(* Schneider Machine Expert - Basic project AWGC_PRODUKSI_TM221CE24R, file version 3.0.0.0 *)
(* ProjectInformations: Name=New project *)

HARDWARE
  Cpu 0: TM221CE24R
  ModuleExtensionObject 0: TM3DI32K
  ModuleExtensionObject 1: TM3AI2H/G
  EthernetConfiguration: NetworkName=M221, IpAllocationMode=FixedAddress, IpAddress=0.0.0.0, SubnetMask=0.0.0.0
  SerialLineConfiguration: Baud=Baud19200, Parity=ParityEven, DataBits=DataBits8, StopBits=StopBits1, PhysicalMedium=PhysicalMediumRs485, TransmissionMode=TransmissionModeModbusRtu, SlaveId=1, Addressing=SlaveAddressing
  MastTask: UsePeriodScanMode=false, PeriodScan=100
  FastTask: Period=255
  CpuBehavior: StartingMode=StartAsPreviousState, AutoSaveRamOnEeprom=true, WatchdogPeriod=250

SYMBOLS  (address, symbol, comment, settings)
  %M0       SYSTEM_ENABLE  "Izin umum gerak"
  %M1       WATER_FAULT  "Fault sinyal level"
  %M2       FAULT_G1  "Fault pintu 1"
  %M3       FAULT_G2  "Fault pintu 2"
  %M4       FAULT_G3  "Fault pintu 3"
  %M5       COMMISSIONING_OK  "Set 1 setelah wiring dan proteksi diuji"
  %M10      REVERSE_G1  "Arah encoder pintu 1 dibalik"
  %M11      REVERSE_G2  "Arah encoder pintu 2 dibalik"
  %M12      REVERSE_G3  "Arah encoder pintu 3 dibalik"
  %M100     G1_BIN_B0  "Binary bit 0 hasil Gray pintu 1"
  %M101     G1_BIN_B1  "Binary bit 1 hasil Gray pintu 1"
  %M102     G1_BIN_B2  "Binary bit 2 hasil Gray pintu 1"
  %M103     G1_BIN_B3  "Binary bit 3 hasil Gray pintu 1"
  %M104     G1_BIN_B4  "Binary bit 4 hasil Gray pintu 1"
  %M105     G1_BIN_B5  "Binary bit 5 hasil Gray pintu 1"
  %M106     G1_BIN_B6  "Binary bit 6 hasil Gray pintu 1"
  %M107     G1_BIN_B7  "Binary bit 7 hasil Gray pintu 1"
  %M110     G2_BIN_B0  "Binary bit 0 hasil Gray pintu 2"
  %M111     G2_BIN_B1  "Binary bit 1 hasil Gray pintu 2"
  %M112     G2_BIN_B2  "Binary bit 2 hasil Gray pintu 2"
  %M113     G2_BIN_B3  "Binary bit 3 hasil Gray pintu 2"
  %M114     G2_BIN_B4  "Binary bit 4 hasil Gray pintu 2"
  %M115     G2_BIN_B5  "Binary bit 5 hasil Gray pintu 2"
  %M116     G2_BIN_B6  "Binary bit 6 hasil Gray pintu 2"
  %M117     G2_BIN_B7  "Binary bit 7 hasil Gray pintu 2"
  %M120     G3_BIN_B0  "Binary bit 0 hasil Gray pintu 3"
  %M121     G3_BIN_B1  "Binary bit 1 hasil Gray pintu 3"
  %M122     G3_BIN_B2  "Binary bit 2 hasil Gray pintu 3"
  %M123     G3_BIN_B3  "Binary bit 3 hasil Gray pintu 3"
  %M124     G3_BIN_B4  "Binary bit 4 hasil Gray pintu 3"
  %M125     G3_BIN_B5  "Binary bit 5 hasil Gray pintu 3"
  %M126     G3_BIN_B6  "Binary bit 6 hasil Gray pintu 3"
  %M127     G3_BIN_B7  "Binary bit 7 hasil Gray pintu 3"
  %M200     AUTO_OPEN_REQ_G1  "Request auto buka G1"
  %M201     AUTO_CLOSE_REQ_G1  "Request auto tutup G1"
  %M202     AUTO_OPEN_REQ_G2  "Request auto buka G2"
  %M203     AUTO_CLOSE_REQ_G2  "Request auto tutup G2"
  %M204     AUTO_OPEN_REQ_G3  "Request auto buka G3"
  %M205     AUTO_CLOSE_REQ_G3  "Request auto tutup G3"
  %M210     MAN_OPEN_REQ_G1  "Request manual buka G1"
  %M211     MAN_CLOSE_REQ_G1  "Request manual tutup G1"
  %M212     MAN_OPEN_REQ_G2  "Request manual buka G2"
  %M213     MAN_CLOSE_REQ_G2  "Request manual tutup G2"
  %M214     MAN_OPEN_REQ_G3  "Request manual buka G3"
  %M215     MAN_CLOSE_REQ_G3  "Request manual tutup G3"
  %M6       SCADA_STOP  "BOOL RW: 1=STOP, 0=release stop; reset to STOP on first RUN"
  %M300     STATUS_I0_0  "Read-only mirror of physical input %I0.0"
  %M301     STATUS_I0_1  "Read-only mirror of physical input %I0.1"
  %M302     STATUS_I0_2  "Read-only mirror of physical input %I0.2"
  %M303     STATUS_I0_3  "Read-only mirror of physical input %I0.3"
  %M304     STATUS_I0_4  "Read-only mirror of physical input %I0.4"
  %M305     STATUS_I0_5  "Read-only mirror of physical input %I0.5"
  %M306     STATUS_I0_6  "Read-only mirror of physical input %I0.6"
  %M307     STATUS_I0_7  "Read-only mirror of physical input %I0.7"
  %M308     STATUS_I0_8  "Read-only mirror of physical input %I0.8"
  %M309     STATUS_I0_9  "Read-only mirror of physical input %I0.9"
  %M310     STATUS_I0_10  "Read-only mirror of physical input %I0.10"
  %M311     STATUS_I0_11  "Read-only mirror of physical input %I0.11"
  %M312     STATUS_I0_12  "Read-only mirror of physical input %I0.12"
  %M313     STATUS_I0_13  "Read-only mirror of physical input %I0.13"
  %M344     STATUS_I1_24  "Read-only mirror of physical input %I1.24"
  %M345     STATUS_I1_25  "Read-only mirror of physical input %I1.25"
  %M346     STATUS_I1_26  "Read-only mirror of physical input %I1.26"
  %M347     STATUS_I1_27  "Read-only mirror of physical input %I1.27"
  %M348     STATUS_I1_28  "Read-only mirror of physical input %I1.28"
  %M349     STATUS_I1_29  "Read-only mirror of physical input %I1.29"
  %M350     STATUS_I1_30  "Read-only mirror of physical input %I1.30"
  %M351     STATUS_I1_31  "Read-only mirror of physical input %I1.31"
  %M360     STATUS_Q0_0  "Read-only mirror of actual output %Q0.0"
  %M361     STATUS_Q0_1  "Read-only mirror of actual output %Q0.1"
  %M362     STATUS_Q0_2  "Read-only mirror of actual output %Q0.2"
  %M363     STATUS_Q0_3  "Read-only mirror of actual output %Q0.3"
  %M364     STATUS_Q0_4  "Read-only mirror of actual output %Q0.4"
  %M365     STATUS_Q0_5  "Read-only mirror of actual output %Q0.5"
  %S13      SB_FIRSTRUN  "Indicates the first controller cycle in RUN mode"
  %MW1      WATER_RANGE_MM  "Range sensor level mm"
  %MW2      LEVEL_RAW_COPY  "Salinan raw input level"
  %MW10     MAX_HEIGHT_G1_MM  "Tinggi maksimum pintu 1 mm"
  %MW11     MAX_HEIGHT_G2_MM  "Tinggi maksimum pintu 2 mm"
  %MW12     MAX_HEIGHT_G3_MM  "Tinggi maksimum pintu 3 mm"
  %MW13     DEADBAND_PCT  "Deadband posisi persen"
  %MW20     ENC_ZERO_G1  "Nilai encoder pintu 1 saat tertutup"
  %MW21     ENC_ZERO_G2  "Nilai encoder pintu 2 saat tertutup"
  %MW22     ENC_ZERO_G3  "Nilai encoder pintu 3 saat tertutup"
  %MW23     ENC_SPAN_G1  "Span count tertutup-terbuka G1"
  %MW24     ENC_SPAN_G2  "Span count tertutup-terbuka G2"
  %MW25     ENC_SPAN_G3  "Span count tertutup-terbuka G3"
  %MW30     ENC_BINARY_G1  "Nilai biner encoder G1"
  %MW31     ENC_BINARY_G2  "Nilai biner encoder G2"
  %MW32     ENC_BINARY_G3  "Nilai biner encoder G3"
  %MW33     POS_COUNT_G1  "Count posisi terkoreksi G1"
  %MW34     POS_COUNT_G2  "Count posisi terkoreksi G2"
  %MW35     POS_COUNT_G3  "Count posisi terkoreksi G3"
  %MW50     TARGET_PCT_G1  "Target bukaan G1 0-100 persen"
  %MW51     TARGET_PCT_G2  "Target bukaan G2 0-100 persen"
  %MW52     TARGET_PCT_G3  "Target bukaan G3 0-100 persen"
  %MW110    SCADA_PROFILE_ID  "221 identifies AWGC SCADA map"
  %MW111    SCADA_PROFILE_VERSION  "3001 production profile: physical inputs and relay outputs"
  %MF60     POSITION_G1_PCT  "Posisi G1 persen"
  %MF62     POSITION_G2_PCT  "Posisi G2 persen"
  %MF64     POSITION_G3_PCT  "Posisi G3 persen"
  %MF66     POSITION_G1_MM  "Posisi G1 mm"
  %MF68     POSITION_G2_MM  "Posisi G2 mm"
  %MF70     POSITION_G3_MM  "Posisi G3 mm"
  %MF72     WATER_LEVEL_MM  "Level air mm"
  %MF74     WATER_LEVEL_PCT  "Level air persen"
  %MF76     WATER_RANGE_REAL  "Range level dalam REAL"
  %MF80     TARGET_G1_REAL  "Target G1 dalam REAL"
  %MF82     TARGET_G2_REAL  "Target G2 dalam REAL"
  %MF84     TARGET_G3_REAL  "Target G3 dalam REAL"
  %MF86     DEADBAND_REAL  "Deadband dalam REAL"
  %MF88     OPEN_THRESHOLD_G1  "Ambang buka G1"
  %MF90     CLOSE_THRESHOLD_G1  "Ambang tutup G1"
  %MF92     OPEN_THRESHOLD_G2  "Ambang buka G2"
  %MF94     CLOSE_THRESHOLD_G2  "Ambang tutup G2"
  %MF96     OPEN_THRESHOLD_G3  "Ambang buka G3"
  %MF98     CLOSE_THRESHOLD_G3  "Ambang tutup G3"
  %I0.0     SAFETY_OK_IN  "Feedback rangkaian safety hardwired sehat"
  %I0.1     LS_CLOSE_G1  "Limit tertutup pintu 1"
  %I0.2     LS_OPEN_G1  "Limit terbuka pintu 1"
  %I0.3     LS_CLOSE_G2  "Limit tertutup pintu 2"
  %I0.4     LS_OPEN_G2  "Limit terbuka pintu 2"
  %I0.5     LS_CLOSE_G3  "Limit tertutup pintu 3"
  %I0.6     LS_OPEN_G3  "Limit terbuka pintu 3"
  %I0.7     OL_OK_G1  "Overload motor pintu 1 sehat"
  %I0.8     OL_OK_G2  "Overload motor pintu 2 sehat"
  %I0.9     OL_OK_G3  "Overload motor pintu 3 sehat"
  %I0.10    SPARE_I010  "Cadangan input"
  %I0.11    SPARE_I011  "Cadangan input"
  %I0.12    SPARE_I012  "Cadangan input"
  %I0.13    SPARE_I013  "Cadangan input"
  %Q0.0     OPEN_G1  "Relay kontaktor OPEN pintu 1"
  %Q0.1     CLOSE_G1  "Relay kontaktor CLOSE pintu 1"
  %Q0.2     OPEN_G2  "Relay kontaktor OPEN pintu 2"
  %Q0.3     CLOSE_G2  "Relay kontaktor CLOSE pintu 2"
  %Q0.4     OPEN_G3  "Relay kontaktor OPEN pintu 3"
  %Q0.5     CLOSE_G3  "Relay kontaktor CLOSE pintu 3"
  %I1.0     ENC_G1_GRAY_B0  "E6CP pintu 1 Gray bit 0"
  %I1.1     ENC_G1_GRAY_B1  "E6CP pintu 1 Gray bit 1"
  %I1.2     ENC_G1_GRAY_B2  "E6CP pintu 1 Gray bit 2"
  %I1.3     ENC_G1_GRAY_B3  "E6CP pintu 1 Gray bit 3"
  %I1.4     ENC_G1_GRAY_B4  "E6CP pintu 1 Gray bit 4"
  %I1.5     ENC_G1_GRAY_B5  "E6CP pintu 1 Gray bit 5"
  %I1.6     ENC_G1_GRAY_B6  "E6CP pintu 1 Gray bit 6"
  %I1.7     ENC_G1_GRAY_B7  "E6CP pintu 1 Gray bit 7"
  %I1.8     ENC_G2_GRAY_B0  "E6CP pintu 2 Gray bit 0"
  %I1.9     ENC_G2_GRAY_B1  "E6CP pintu 2 Gray bit 1"
  %I1.10    ENC_G2_GRAY_B2  "E6CP pintu 2 Gray bit 2"
  %I1.11    ENC_G2_GRAY_B3  "E6CP pintu 2 Gray bit 3"
  %I1.12    ENC_G2_GRAY_B4  "E6CP pintu 2 Gray bit 4"
  %I1.13    ENC_G2_GRAY_B5  "E6CP pintu 2 Gray bit 5"
  %I1.14    ENC_G2_GRAY_B6  "E6CP pintu 2 Gray bit 6"
  %I1.15    ENC_G2_GRAY_B7  "E6CP pintu 2 Gray bit 7"
  %I1.16    ENC_G3_GRAY_B0  "E6CP pintu 3 Gray bit 0"
  %I1.17    ENC_G3_GRAY_B1  "E6CP pintu 3 Gray bit 1"
  %I1.18    ENC_G3_GRAY_B2  "E6CP pintu 3 Gray bit 2"
  %I1.19    ENC_G3_GRAY_B3  "E6CP pintu 3 Gray bit 3"
  %I1.20    ENC_G3_GRAY_B4  "E6CP pintu 3 Gray bit 4"
  %I1.21    ENC_G3_GRAY_B5  "E6CP pintu 3 Gray bit 5"
  %I1.22    ENC_G3_GRAY_B6  "E6CP pintu 3 Gray bit 6"
  %I1.23    ENC_G3_GRAY_B7  "E6CP pintu 3 Gray bit 7"
  %I1.24    MODE_AUTO  "Selector 1=AUTO 0=MANUAL"
  %I1.25    MAN_OPEN_G1  "PB manual buka pintu 1"
  %I1.26    MAN_CLOSE_G1  "PB manual tutup pintu 1"
  %I1.27    MAN_OPEN_G2  "PB manual buka pintu 2"
  %I1.28    MAN_CLOSE_G2  "PB manual tutup pintu 2"
  %I1.29    MAN_OPEN_G3  "PB manual buka pintu 3"
  %I1.30    MAN_CLOSE_G3  "PB manual tutup pintu 3"
  %I1.31    RESET_FAULT  "PB reset fault"
  %IW2.0    LEVEL_RAW  "Sensor level 4-20 mA raw 4000-20000"  [Type=Type_4_20mA, Scope=Scope_Customized, Minimum=4000, Maximum=20000]

POU AWGC_3_PINTU_IL
  (* SectionNumber=1 *)

// Rung 0: REV3_SCADA_VERSION
// SCADA compatibility marker for production profile.
  LD 1
  [ %MW111 := 3001 ]      (* SCADA_PROFILE_VERSION *)
  // as ST:
  //   SCADA_PROFILE_VERSION := 3001;

// Rung 1: REV3_SCADA_ID
// SCADA compatibility marker for production profile.
  LD 1
  [ %MW110 := 221 ]       (* SCADA_PROFILE_ID *)
  // as ST:
  //   SCADA_PROFILE_ID := 221;

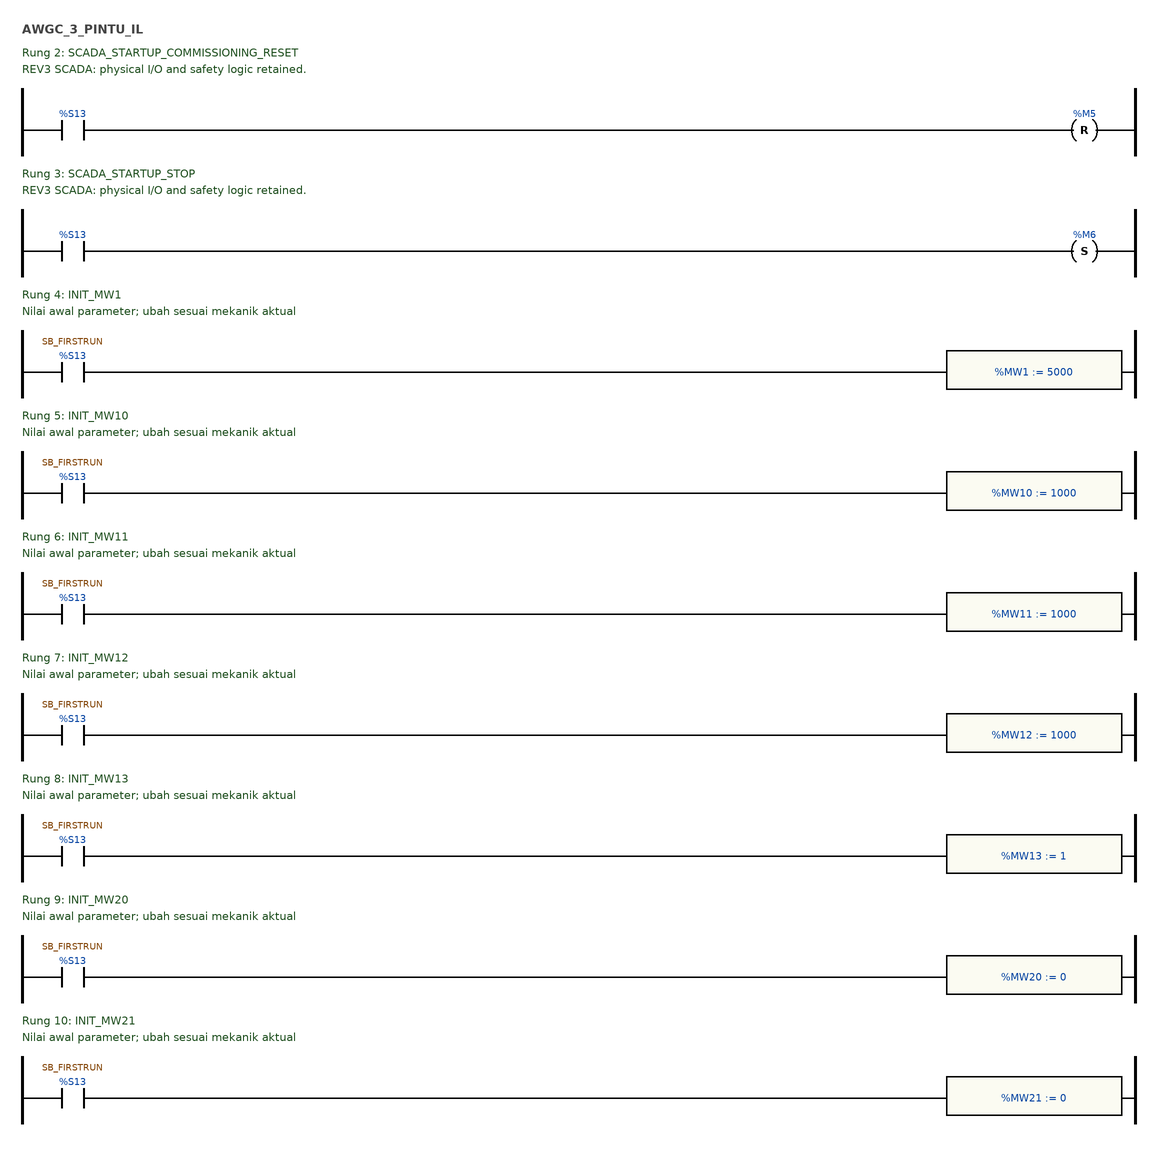

// Rung 2: SCADA_STARTUP_COMMISSIONING_RESET
// REV3 SCADA: physical I/O and safety logic retained.
  LD %S13                 (* SB_FIRSTRUN *)
  R %M5                   (* COMMISSIONING_OK *)
  // as ST:
  //   IF SB_FIRSTRUN THEN COMMISSIONING_OK := FALSE; END_IF;

// Rung 3: SCADA_STARTUP_STOP
// REV3 SCADA: physical I/O and safety logic retained.
  LD %S13                 (* SB_FIRSTRUN *)
  S %M6                   (* SCADA_STOP *)
  // as ST:
  //   IF SB_FIRSTRUN THEN SCADA_STOP := TRUE; END_IF;

// Rung 4: INIT_MW1
// Nilai awal parameter; ubah sesuai mekanik aktual
  LD %S13                 (* SB_FIRSTRUN *)
  [ %MW1 := 5000 ]        (* WATER_RANGE_MM *)
  // as ST:
  //   IF SB_FIRSTRUN THEN WATER_RANGE_MM := 5000; END_IF;

// Rung 5: INIT_MW10
// Nilai awal parameter; ubah sesuai mekanik aktual
  LD %S13                 (* SB_FIRSTRUN *)
  [ %MW10 := 1000 ]       (* MAX_HEIGHT_G1_MM *)
  // as ST:
  //   IF SB_FIRSTRUN THEN MAX_HEIGHT_G1_MM := 1000; END_IF;

// Rung 6: INIT_MW11
// Nilai awal parameter; ubah sesuai mekanik aktual
  LD %S13                 (* SB_FIRSTRUN *)
  [ %MW11 := 1000 ]       (* MAX_HEIGHT_G2_MM *)
  // as ST:
  //   IF SB_FIRSTRUN THEN MAX_HEIGHT_G2_MM := 1000; END_IF;

// Rung 7: INIT_MW12
// Nilai awal parameter; ubah sesuai mekanik aktual
  LD %S13                 (* SB_FIRSTRUN *)
  [ %MW12 := 1000 ]       (* MAX_HEIGHT_G3_MM *)
  // as ST:
  //   IF SB_FIRSTRUN THEN MAX_HEIGHT_G3_MM := 1000; END_IF;

// Rung 8: INIT_MW13
// Nilai awal parameter; ubah sesuai mekanik aktual
  LD %S13                 (* SB_FIRSTRUN *)
  [ %MW13 := 1 ]          (* DEADBAND_PCT *)
  // as ST:
  //   IF SB_FIRSTRUN THEN DEADBAND_PCT := 1; END_IF;

// Rung 9: INIT_MW20
// Nilai awal parameter; ubah sesuai mekanik aktual
  LD %S13                 (* SB_FIRSTRUN *)
  [ %MW20 := 0 ]          (* ENC_ZERO_G1 *)
  // as ST:
  //   IF SB_FIRSTRUN THEN ENC_ZERO_G1 := 0; END_IF;

// Rung 10: INIT_MW21
// Nilai awal parameter; ubah sesuai mekanik aktual
  LD %S13                 (* SB_FIRSTRUN *)
  [ %MW21 := 0 ]          (* ENC_ZERO_G2 *)
  // as ST:
  //   IF SB_FIRSTRUN THEN ENC_ZERO_G2 := 0; END_IF;

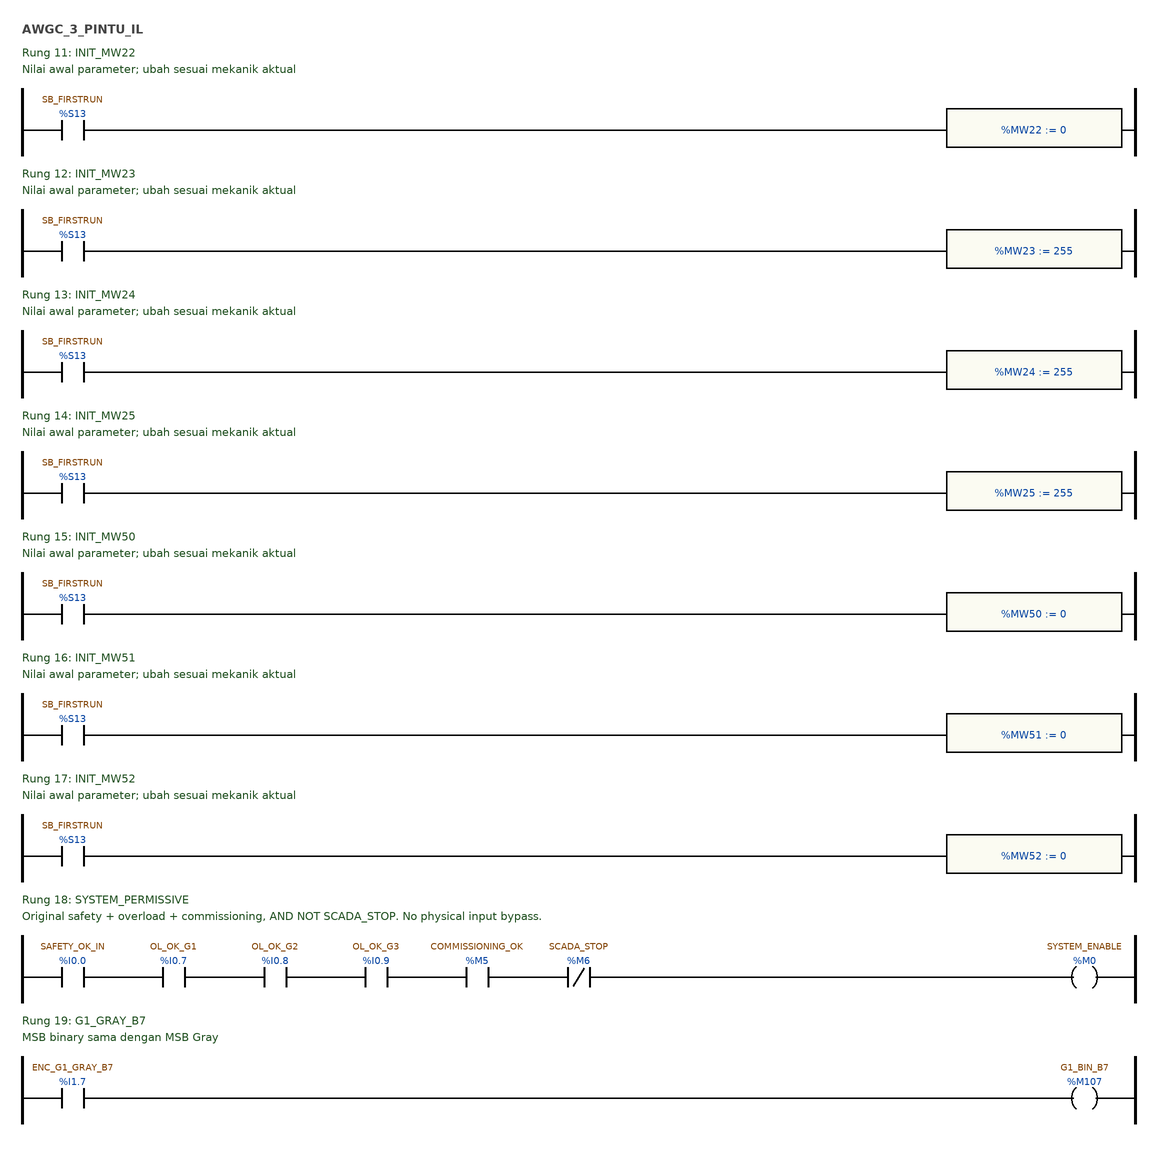

// Rung 11: INIT_MW22
// Nilai awal parameter; ubah sesuai mekanik aktual
  LD %S13                 (* SB_FIRSTRUN *)
  [ %MW22 := 0 ]          (* ENC_ZERO_G3 *)
  // as ST:
  //   IF SB_FIRSTRUN THEN ENC_ZERO_G3 := 0; END_IF;

// Rung 12: INIT_MW23
// Nilai awal parameter; ubah sesuai mekanik aktual
  LD %S13                 (* SB_FIRSTRUN *)
  [ %MW23 := 255 ]        (* ENC_SPAN_G1 *)
  // as ST:
  //   IF SB_FIRSTRUN THEN ENC_SPAN_G1 := 255; END_IF;

// Rung 13: INIT_MW24
// Nilai awal parameter; ubah sesuai mekanik aktual
  LD %S13                 (* SB_FIRSTRUN *)
  [ %MW24 := 255 ]        (* ENC_SPAN_G2 *)
  // as ST:
  //   IF SB_FIRSTRUN THEN ENC_SPAN_G2 := 255; END_IF;

// Rung 14: INIT_MW25
// Nilai awal parameter; ubah sesuai mekanik aktual
  LD %S13                 (* SB_FIRSTRUN *)
  [ %MW25 := 255 ]        (* ENC_SPAN_G3 *)
  // as ST:
  //   IF SB_FIRSTRUN THEN ENC_SPAN_G3 := 255; END_IF;

// Rung 15: INIT_MW50
// Nilai awal parameter; ubah sesuai mekanik aktual
  LD %S13                 (* SB_FIRSTRUN *)
  [ %MW50 := 0 ]          (* TARGET_PCT_G1 *)
  // as ST:
  //   IF SB_FIRSTRUN THEN TARGET_PCT_G1 := 0; END_IF;

// Rung 16: INIT_MW51
// Nilai awal parameter; ubah sesuai mekanik aktual
  LD %S13                 (* SB_FIRSTRUN *)
  [ %MW51 := 0 ]          (* TARGET_PCT_G2 *)
  // as ST:
  //   IF SB_FIRSTRUN THEN TARGET_PCT_G2 := 0; END_IF;

// Rung 17: INIT_MW52
// Nilai awal parameter; ubah sesuai mekanik aktual
  LD %S13                 (* SB_FIRSTRUN *)
  [ %MW52 := 0 ]          (* TARGET_PCT_G3 *)
  // as ST:
  //   IF SB_FIRSTRUN THEN TARGET_PCT_G3 := 0; END_IF;

// Rung 18: SYSTEM_PERMISSIVE
// Original safety + overload + commissioning, AND NOT SCADA_STOP. No physical input bypass.
  LD %I0.0                (* SAFETY_OK_IN *)
  AND %I0.7               (* OL_OK_G1 *)
  AND %I0.8               (* OL_OK_G2 *)
  AND %I0.9               (* OL_OK_G3 *)
  AND %M5                 (* COMMISSIONING_OK *)
  ANDN %M6                (* SCADA_STOP *)
  ST %M0                  (* SYSTEM_ENABLE *)
  // %M6: 1=STOP; startup STOP. This is not an emergency stop.
  // as ST:
  //   SYSTEM_ENABLE := SAFETY_OK_IN AND OL_OK_G1 AND OL_OK_G2 AND OL_OK_G3 AND COMMISSIONING_OK AND NOT SCADA_STOP;

// Rung 19: G1_GRAY_B7
// MSB binary sama dengan MSB Gray
  LD %I1.7                (* ENC_G1_GRAY_B7 *)
  ST %M107                (* G1_BIN_B7 *)
  // as ST:
  //   G1_BIN_B7 := ENC_G1_GRAY_B7;

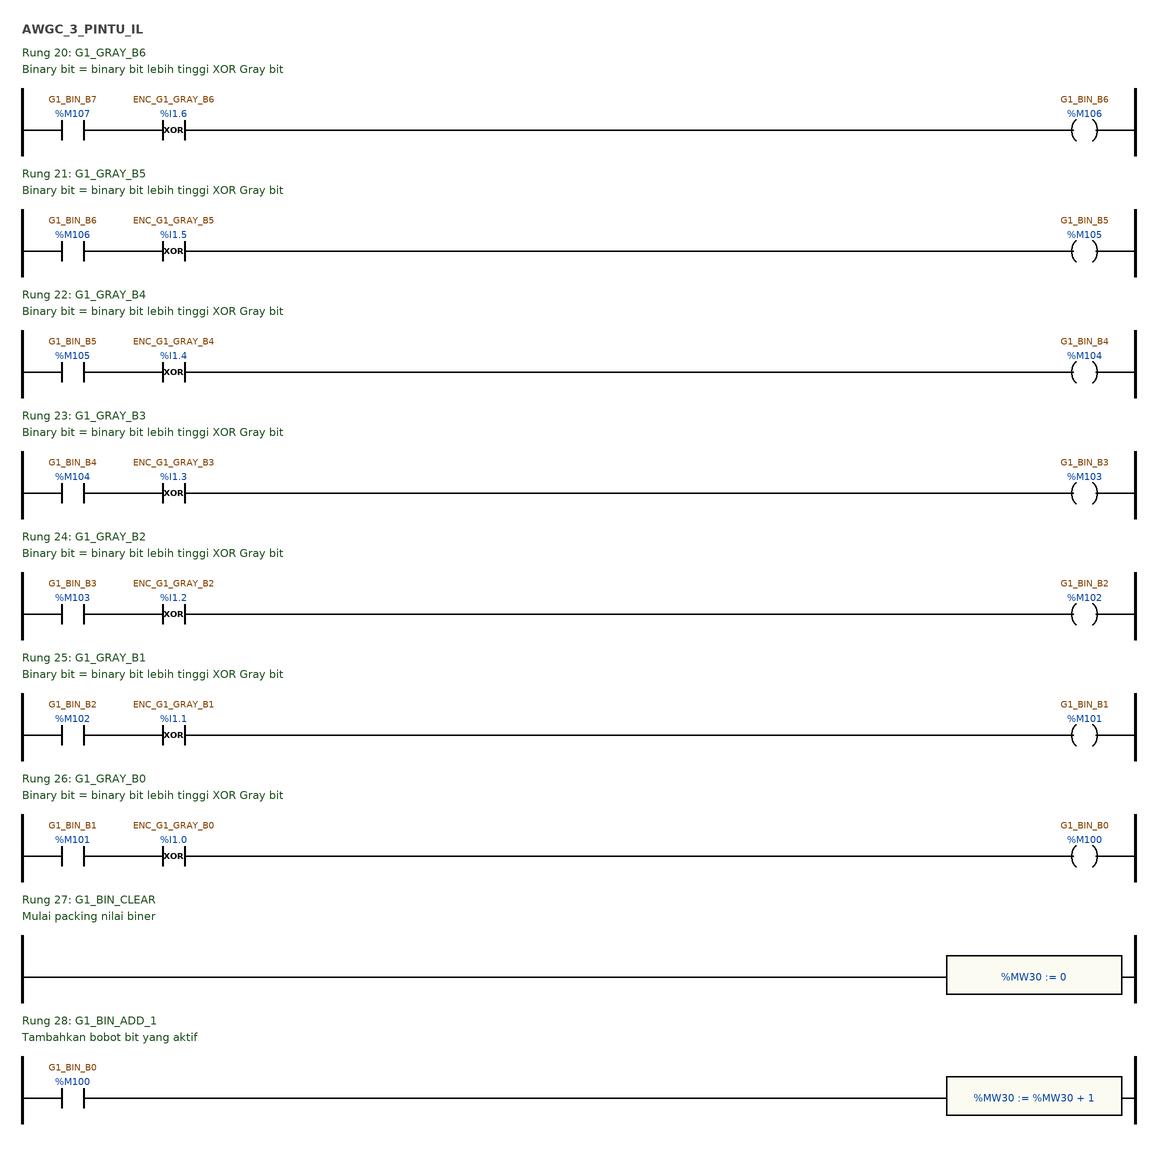

// Rung 20: G1_GRAY_B6
// Binary bit = binary bit lebih tinggi XOR Gray bit
  LD %M107                (* G1_BIN_B7 *)
  XOR %I1.6               (* ENC_G1_GRAY_B6 *)
  ST %M106                (* G1_BIN_B6 *)
  // as ST:
  //   G1_BIN_B6 := G1_BIN_B7 XOR ENC_G1_GRAY_B6;

// Rung 21: G1_GRAY_B5
// Binary bit = binary bit lebih tinggi XOR Gray bit
  LD %M106                (* G1_BIN_B6 *)
  XOR %I1.5               (* ENC_G1_GRAY_B5 *)
  ST %M105                (* G1_BIN_B5 *)
  // as ST:
  //   G1_BIN_B5 := G1_BIN_B6 XOR ENC_G1_GRAY_B5;

// Rung 22: G1_GRAY_B4
// Binary bit = binary bit lebih tinggi XOR Gray bit
  LD %M105                (* G1_BIN_B5 *)
  XOR %I1.4               (* ENC_G1_GRAY_B4 *)
  ST %M104                (* G1_BIN_B4 *)
  // as ST:
  //   G1_BIN_B4 := G1_BIN_B5 XOR ENC_G1_GRAY_B4;

// Rung 23: G1_GRAY_B3
// Binary bit = binary bit lebih tinggi XOR Gray bit
  LD %M104                (* G1_BIN_B4 *)
  XOR %I1.3               (* ENC_G1_GRAY_B3 *)
  ST %M103                (* G1_BIN_B3 *)
  // as ST:
  //   G1_BIN_B3 := G1_BIN_B4 XOR ENC_G1_GRAY_B3;

// Rung 24: G1_GRAY_B2
// Binary bit = binary bit lebih tinggi XOR Gray bit
  LD %M103                (* G1_BIN_B3 *)
  XOR %I1.2               (* ENC_G1_GRAY_B2 *)
  ST %M102                (* G1_BIN_B2 *)
  // as ST:
  //   G1_BIN_B2 := G1_BIN_B3 XOR ENC_G1_GRAY_B2;

// Rung 25: G1_GRAY_B1
// Binary bit = binary bit lebih tinggi XOR Gray bit
  LD %M102                (* G1_BIN_B2 *)
  XOR %I1.1               (* ENC_G1_GRAY_B1 *)
  ST %M101                (* G1_BIN_B1 *)
  // as ST:
  //   G1_BIN_B1 := G1_BIN_B2 XOR ENC_G1_GRAY_B1;

// Rung 26: G1_GRAY_B0
// Binary bit = binary bit lebih tinggi XOR Gray bit
  LD %M101                (* G1_BIN_B1 *)
  XOR %I1.0               (* ENC_G1_GRAY_B0 *)
  ST %M100                (* G1_BIN_B0 *)
  // as ST:
  //   G1_BIN_B0 := G1_BIN_B1 XOR ENC_G1_GRAY_B0;

// Rung 27: G1_BIN_CLEAR
// Mulai packing nilai biner
  LD 1
  [ %MW30 := 0 ]          (* ENC_BINARY_G1 *)
  // as ST:
  //   ENC_BINARY_G1 := 0;

// Rung 28: G1_BIN_ADD_1
// Tambahkan bobot bit yang aktif
  LD %M100                (* G1_BIN_B0 *)
  [ %MW30 := %MW30 + 1 ]  (* ENC_BINARY_G1, ENC_BINARY_G1 *)
  // as ST:
  //   IF G1_BIN_B0 THEN ENC_BINARY_G1 := ENC_BINARY_G1 + 1; END_IF;

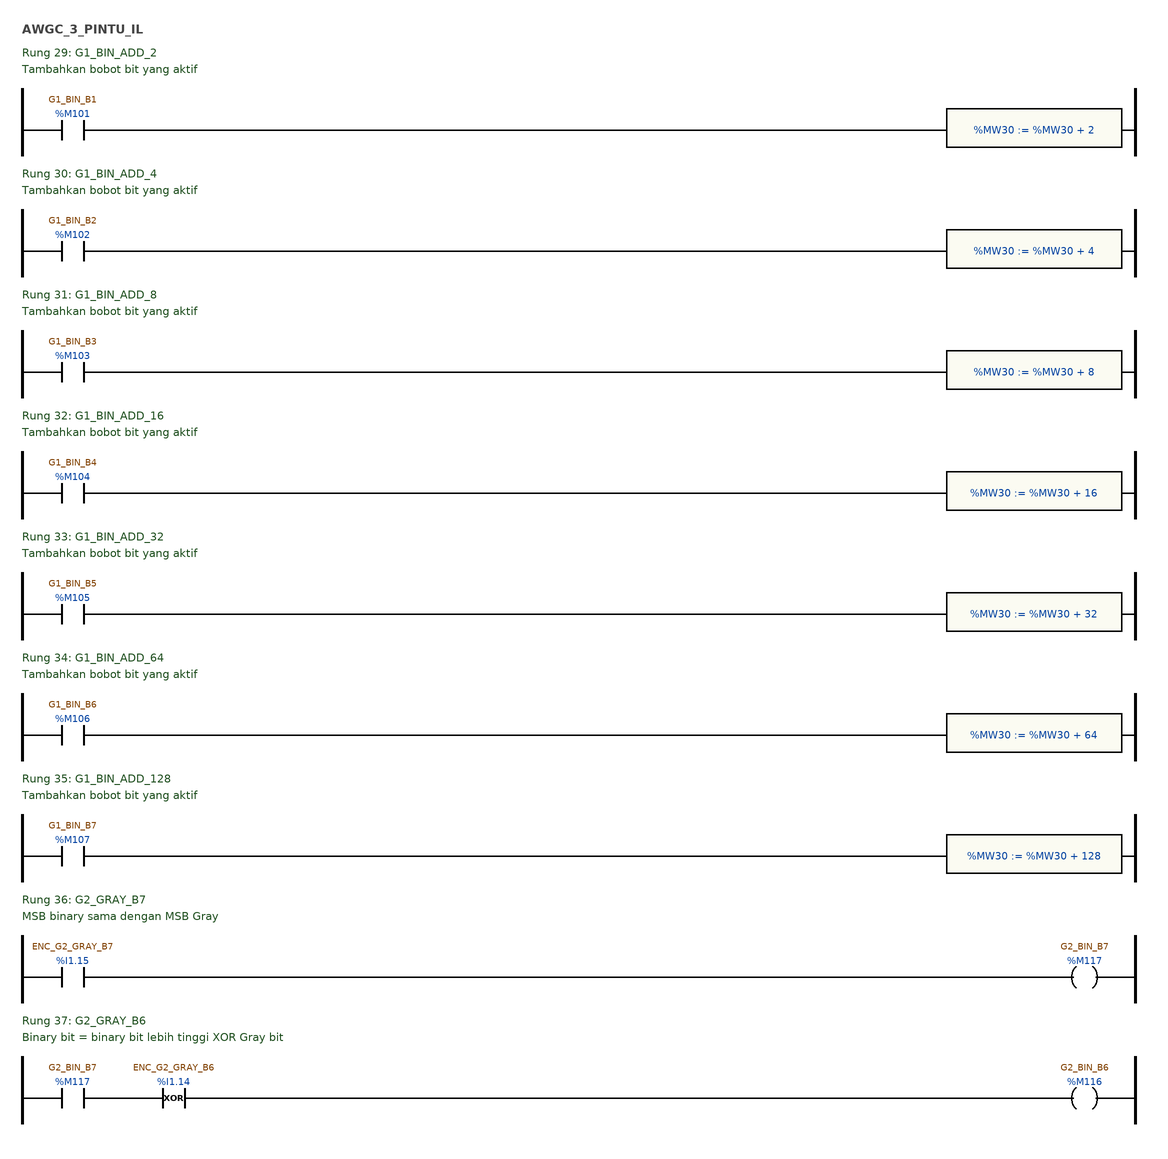

// Rung 29: G1_BIN_ADD_2
// Tambahkan bobot bit yang aktif
  LD %M101                (* G1_BIN_B1 *)
  [ %MW30 := %MW30 + 2 ]  (* ENC_BINARY_G1, ENC_BINARY_G1 *)
  // as ST:
  //   IF G1_BIN_B1 THEN ENC_BINARY_G1 := ENC_BINARY_G1 + 2; END_IF;

// Rung 30: G1_BIN_ADD_4
// Tambahkan bobot bit yang aktif
  LD %M102                (* G1_BIN_B2 *)
  [ %MW30 := %MW30 + 4 ]  (* ENC_BINARY_G1, ENC_BINARY_G1 *)
  // as ST:
  //   IF G1_BIN_B2 THEN ENC_BINARY_G1 := ENC_BINARY_G1 + 4; END_IF;

// Rung 31: G1_BIN_ADD_8
// Tambahkan bobot bit yang aktif
  LD %M103                (* G1_BIN_B3 *)
  [ %MW30 := %MW30 + 8 ]  (* ENC_BINARY_G1, ENC_BINARY_G1 *)
  // as ST:
  //   IF G1_BIN_B3 THEN ENC_BINARY_G1 := ENC_BINARY_G1 + 8; END_IF;

// Rung 32: G1_BIN_ADD_16
// Tambahkan bobot bit yang aktif
  LD %M104                (* G1_BIN_B4 *)
  [ %MW30 := %MW30 + 16 ] (* ENC_BINARY_G1, ENC_BINARY_G1 *)
  // as ST:
  //   IF G1_BIN_B4 THEN ENC_BINARY_G1 := ENC_BINARY_G1 + 16; END_IF;

// Rung 33: G1_BIN_ADD_32
// Tambahkan bobot bit yang aktif
  LD %M105                (* G1_BIN_B5 *)
  [ %MW30 := %MW30 + 32 ] (* ENC_BINARY_G1, ENC_BINARY_G1 *)
  // as ST:
  //   IF G1_BIN_B5 THEN ENC_BINARY_G1 := ENC_BINARY_G1 + 32; END_IF;

// Rung 34: G1_BIN_ADD_64
// Tambahkan bobot bit yang aktif
  LD %M106                (* G1_BIN_B6 *)
  [ %MW30 := %MW30 + 64 ] (* ENC_BINARY_G1, ENC_BINARY_G1 *)
  // as ST:
  //   IF G1_BIN_B6 THEN ENC_BINARY_G1 := ENC_BINARY_G1 + 64; END_IF;

// Rung 35: G1_BIN_ADD_128
// Tambahkan bobot bit yang aktif
  LD %M107                (* G1_BIN_B7 *)
  [ %MW30 := %MW30 + 128 ](* ENC_BINARY_G1, ENC_BINARY_G1 *)
  // as ST:
  //   IF G1_BIN_B7 THEN ENC_BINARY_G1 := ENC_BINARY_G1 + 128; END_IF;

// Rung 36: G2_GRAY_B7
// MSB binary sama dengan MSB Gray
  LD %I1.15               (* ENC_G2_GRAY_B7 *)
  ST %M117                (* G2_BIN_B7 *)
  // as ST:
  //   G2_BIN_B7 := ENC_G2_GRAY_B7;

// Rung 37: G2_GRAY_B6
// Binary bit = binary bit lebih tinggi XOR Gray bit
  LD %M117                (* G2_BIN_B7 *)
  XOR %I1.14              (* ENC_G2_GRAY_B6 *)
  ST %M116                (* G2_BIN_B6 *)
  // as ST:
  //   G2_BIN_B6 := G2_BIN_B7 XOR ENC_G2_GRAY_B6;

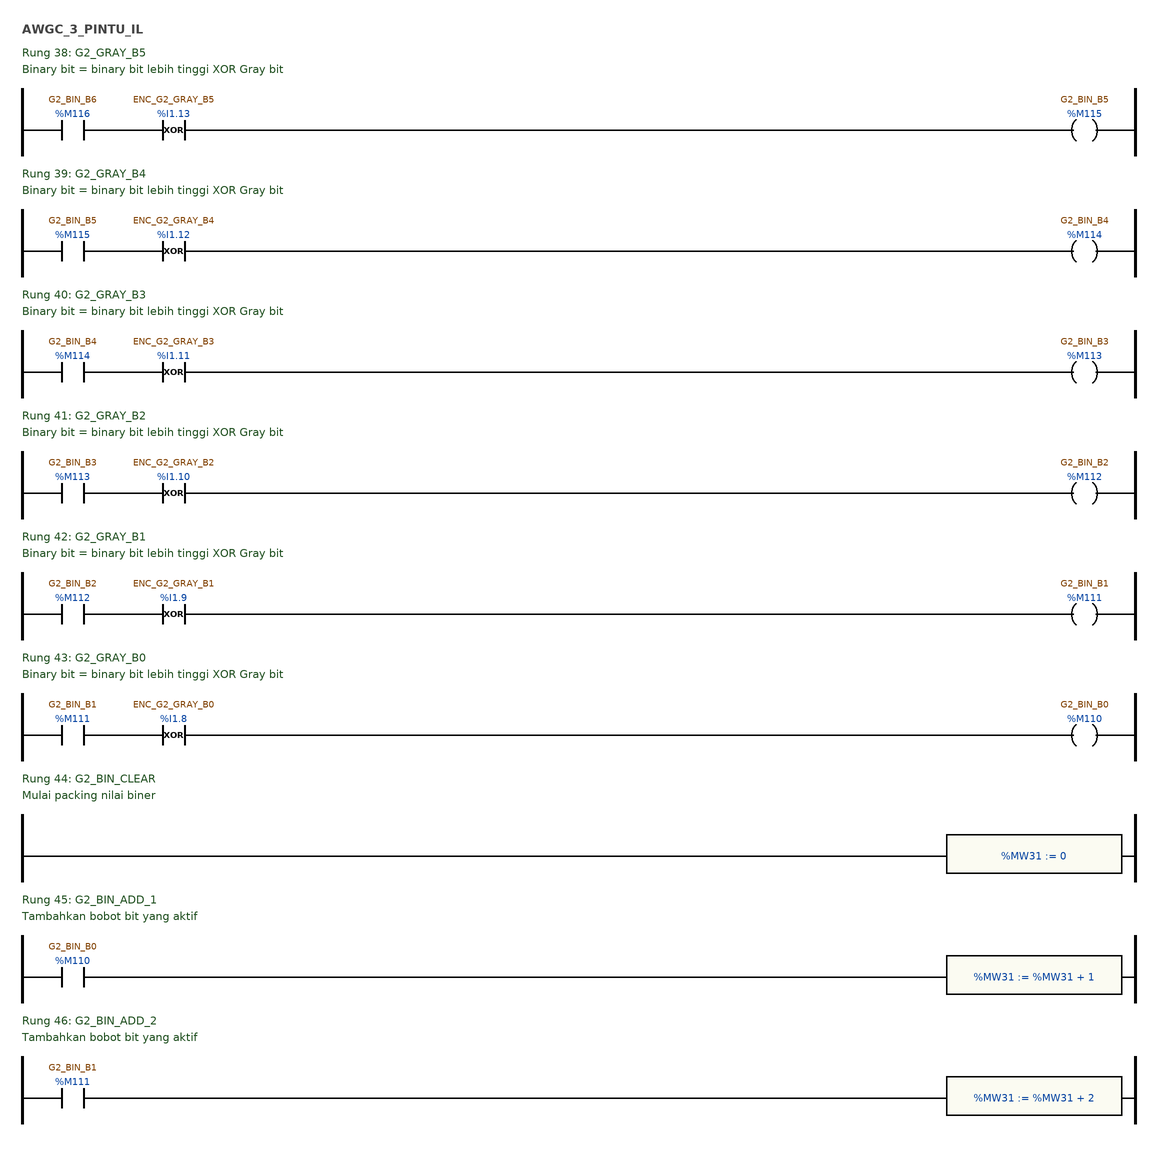

// Rung 38: G2_GRAY_B5
// Binary bit = binary bit lebih tinggi XOR Gray bit
  LD %M116                (* G2_BIN_B6 *)
  XOR %I1.13              (* ENC_G2_GRAY_B5 *)
  ST %M115                (* G2_BIN_B5 *)
  // as ST:
  //   G2_BIN_B5 := G2_BIN_B6 XOR ENC_G2_GRAY_B5;

// Rung 39: G2_GRAY_B4
// Binary bit = binary bit lebih tinggi XOR Gray bit
  LD %M115                (* G2_BIN_B5 *)
  XOR %I1.12              (* ENC_G2_GRAY_B4 *)
  ST %M114                (* G2_BIN_B4 *)
  // as ST:
  //   G2_BIN_B4 := G2_BIN_B5 XOR ENC_G2_GRAY_B4;

// Rung 40: G2_GRAY_B3
// Binary bit = binary bit lebih tinggi XOR Gray bit
  LD %M114                (* G2_BIN_B4 *)
  XOR %I1.11              (* ENC_G2_GRAY_B3 *)
  ST %M113                (* G2_BIN_B3 *)
  // as ST:
  //   G2_BIN_B3 := G2_BIN_B4 XOR ENC_G2_GRAY_B3;

// Rung 41: G2_GRAY_B2
// Binary bit = binary bit lebih tinggi XOR Gray bit
  LD %M113                (* G2_BIN_B3 *)
  XOR %I1.10              (* ENC_G2_GRAY_B2 *)
  ST %M112                (* G2_BIN_B2 *)
  // as ST:
  //   G2_BIN_B2 := G2_BIN_B3 XOR ENC_G2_GRAY_B2;

// Rung 42: G2_GRAY_B1
// Binary bit = binary bit lebih tinggi XOR Gray bit
  LD %M112                (* G2_BIN_B2 *)
  XOR %I1.9               (* ENC_G2_GRAY_B1 *)
  ST %M111                (* G2_BIN_B1 *)
  // as ST:
  //   G2_BIN_B1 := G2_BIN_B2 XOR ENC_G2_GRAY_B1;

// Rung 43: G2_GRAY_B0
// Binary bit = binary bit lebih tinggi XOR Gray bit
  LD %M111                (* G2_BIN_B1 *)
  XOR %I1.8               (* ENC_G2_GRAY_B0 *)
  ST %M110                (* G2_BIN_B0 *)
  // as ST:
  //   G2_BIN_B0 := G2_BIN_B1 XOR ENC_G2_GRAY_B0;

// Rung 44: G2_BIN_CLEAR
// Mulai packing nilai biner
  LD 1
  [ %MW31 := 0 ]          (* ENC_BINARY_G2 *)
  // as ST:
  //   ENC_BINARY_G2 := 0;

// Rung 45: G2_BIN_ADD_1
// Tambahkan bobot bit yang aktif
  LD %M110                (* G2_BIN_B0 *)
  [ %MW31 := %MW31 + 1 ]  (* ENC_BINARY_G2, ENC_BINARY_G2 *)
  // as ST:
  //   IF G2_BIN_B0 THEN ENC_BINARY_G2 := ENC_BINARY_G2 + 1; END_IF;

// Rung 46: G2_BIN_ADD_2
// Tambahkan bobot bit yang aktif
  LD %M111                (* G2_BIN_B1 *)
  [ %MW31 := %MW31 + 2 ]  (* ENC_BINARY_G2, ENC_BINARY_G2 *)
  // as ST:
  //   IF G2_BIN_B1 THEN ENC_BINARY_G2 := ENC_BINARY_G2 + 2; END_IF;

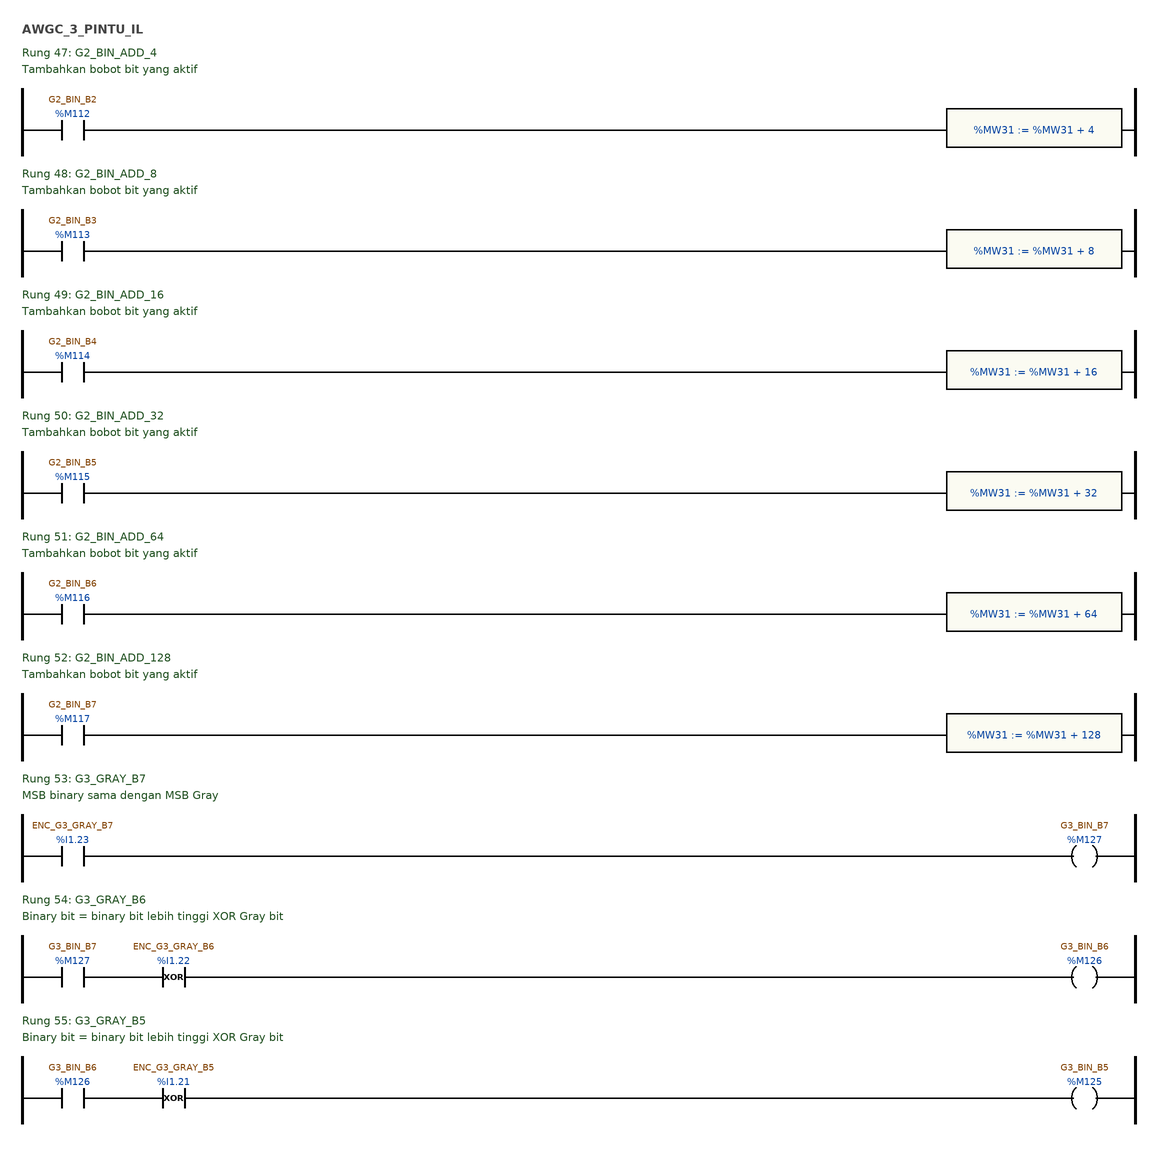

// Rung 47: G2_BIN_ADD_4
// Tambahkan bobot bit yang aktif
  LD %M112                (* G2_BIN_B2 *)
  [ %MW31 := %MW31 + 4 ]  (* ENC_BINARY_G2, ENC_BINARY_G2 *)
  // as ST:
  //   IF G2_BIN_B2 THEN ENC_BINARY_G2 := ENC_BINARY_G2 + 4; END_IF;

// Rung 48: G2_BIN_ADD_8
// Tambahkan bobot bit yang aktif
  LD %M113                (* G2_BIN_B3 *)
  [ %MW31 := %MW31 + 8 ]  (* ENC_BINARY_G2, ENC_BINARY_G2 *)
  // as ST:
  //   IF G2_BIN_B3 THEN ENC_BINARY_G2 := ENC_BINARY_G2 + 8; END_IF;

// Rung 49: G2_BIN_ADD_16
// Tambahkan bobot bit yang aktif
  LD %M114                (* G2_BIN_B4 *)
  [ %MW31 := %MW31 + 16 ] (* ENC_BINARY_G2, ENC_BINARY_G2 *)
  // as ST:
  //   IF G2_BIN_B4 THEN ENC_BINARY_G2 := ENC_BINARY_G2 + 16; END_IF;

// Rung 50: G2_BIN_ADD_32
// Tambahkan bobot bit yang aktif
  LD %M115                (* G2_BIN_B5 *)
  [ %MW31 := %MW31 + 32 ] (* ENC_BINARY_G2, ENC_BINARY_G2 *)
  // as ST:
  //   IF G2_BIN_B5 THEN ENC_BINARY_G2 := ENC_BINARY_G2 + 32; END_IF;

// Rung 51: G2_BIN_ADD_64
// Tambahkan bobot bit yang aktif
  LD %M116                (* G2_BIN_B6 *)
  [ %MW31 := %MW31 + 64 ] (* ENC_BINARY_G2, ENC_BINARY_G2 *)
  // as ST:
  //   IF G2_BIN_B6 THEN ENC_BINARY_G2 := ENC_BINARY_G2 + 64; END_IF;

// Rung 52: G2_BIN_ADD_128
// Tambahkan bobot bit yang aktif
  LD %M117                (* G2_BIN_B7 *)
  [ %MW31 := %MW31 + 128 ](* ENC_BINARY_G2, ENC_BINARY_G2 *)
  // as ST:
  //   IF G2_BIN_B7 THEN ENC_BINARY_G2 := ENC_BINARY_G2 + 128; END_IF;

// Rung 53: G3_GRAY_B7
// MSB binary sama dengan MSB Gray
  LD %I1.23               (* ENC_G3_GRAY_B7 *)
  ST %M127                (* G3_BIN_B7 *)
  // as ST:
  //   G3_BIN_B7 := ENC_G3_GRAY_B7;

// Rung 54: G3_GRAY_B6
// Binary bit = binary bit lebih tinggi XOR Gray bit
  LD %M127                (* G3_BIN_B7 *)
  XOR %I1.22              (* ENC_G3_GRAY_B6 *)
  ST %M126                (* G3_BIN_B6 *)
  // as ST:
  //   G3_BIN_B6 := G3_BIN_B7 XOR ENC_G3_GRAY_B6;

// Rung 55: G3_GRAY_B5
// Binary bit = binary bit lebih tinggi XOR Gray bit
  LD %M126                (* G3_BIN_B6 *)
  XOR %I1.21              (* ENC_G3_GRAY_B5 *)
  ST %M125                (* G3_BIN_B5 *)
  // as ST:
  //   G3_BIN_B5 := G3_BIN_B6 XOR ENC_G3_GRAY_B5;

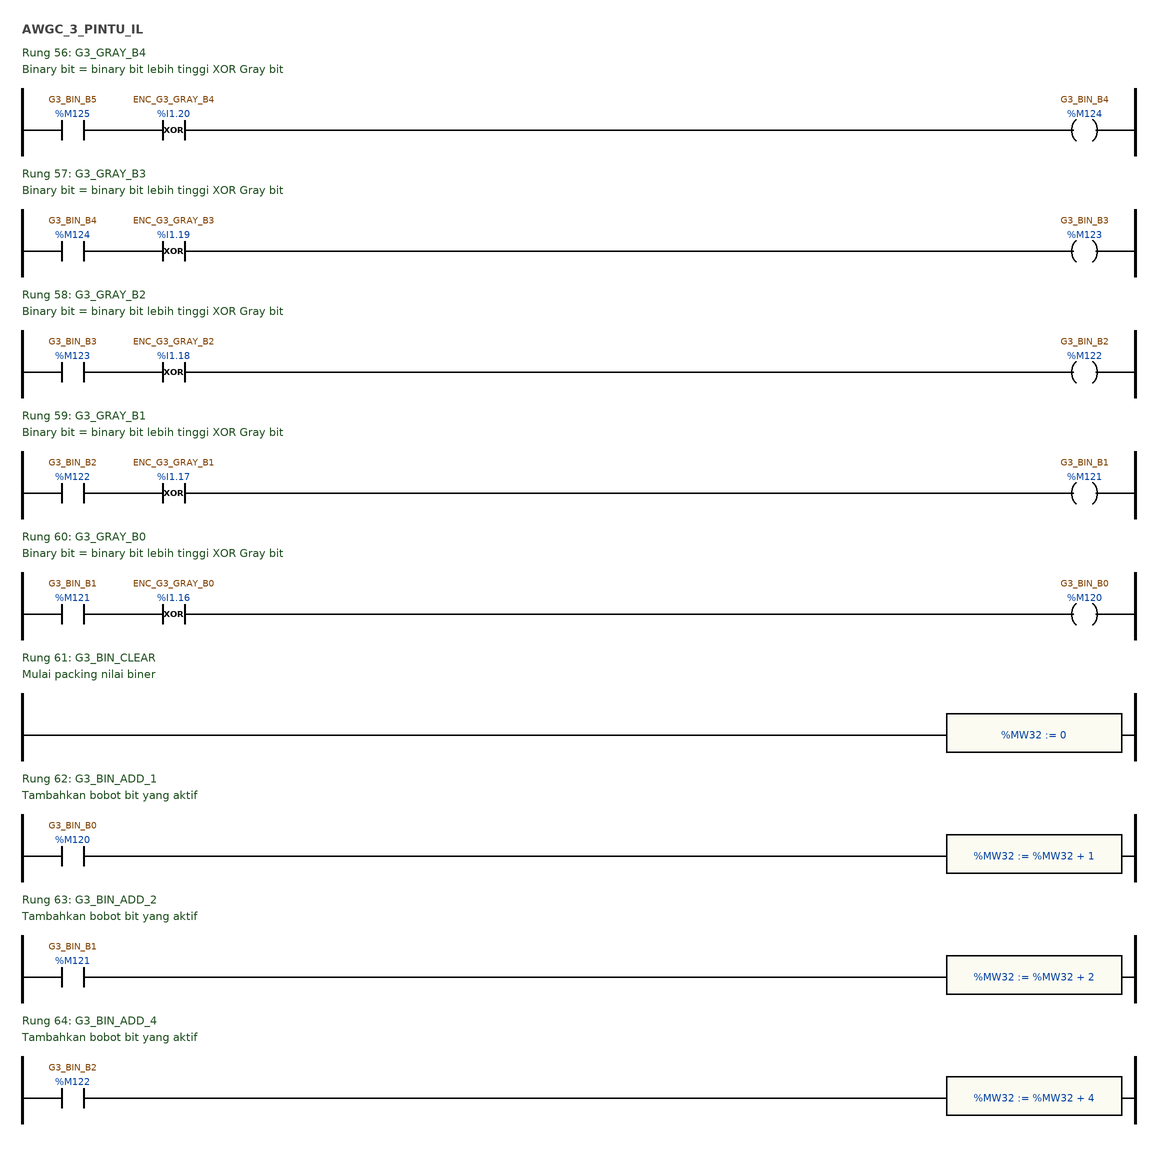

// Rung 56: G3_GRAY_B4
// Binary bit = binary bit lebih tinggi XOR Gray bit
  LD %M125                (* G3_BIN_B5 *)
  XOR %I1.20              (* ENC_G3_GRAY_B4 *)
  ST %M124                (* G3_BIN_B4 *)
  // as ST:
  //   G3_BIN_B4 := G3_BIN_B5 XOR ENC_G3_GRAY_B4;

// Rung 57: G3_GRAY_B3
// Binary bit = binary bit lebih tinggi XOR Gray bit
  LD %M124                (* G3_BIN_B4 *)
  XOR %I1.19              (* ENC_G3_GRAY_B3 *)
  ST %M123                (* G3_BIN_B3 *)
  // as ST:
  //   G3_BIN_B3 := G3_BIN_B4 XOR ENC_G3_GRAY_B3;

// Rung 58: G3_GRAY_B2
// Binary bit = binary bit lebih tinggi XOR Gray bit
  LD %M123                (* G3_BIN_B3 *)
  XOR %I1.18              (* ENC_G3_GRAY_B2 *)
  ST %M122                (* G3_BIN_B2 *)
  // as ST:
  //   G3_BIN_B2 := G3_BIN_B3 XOR ENC_G3_GRAY_B2;

// Rung 59: G3_GRAY_B1
// Binary bit = binary bit lebih tinggi XOR Gray bit
  LD %M122                (* G3_BIN_B2 *)
  XOR %I1.17              (* ENC_G3_GRAY_B1 *)
  ST %M121                (* G3_BIN_B1 *)
  // as ST:
  //   G3_BIN_B1 := G3_BIN_B2 XOR ENC_G3_GRAY_B1;

// Rung 60: G3_GRAY_B0
// Binary bit = binary bit lebih tinggi XOR Gray bit
  LD %M121                (* G3_BIN_B1 *)
  XOR %I1.16              (* ENC_G3_GRAY_B0 *)
  ST %M120                (* G3_BIN_B0 *)
  // as ST:
  //   G3_BIN_B0 := G3_BIN_B1 XOR ENC_G3_GRAY_B0;

// Rung 61: G3_BIN_CLEAR
// Mulai packing nilai biner
  LD 1
  [ %MW32 := 0 ]          (* ENC_BINARY_G3 *)
  // as ST:
  //   ENC_BINARY_G3 := 0;

// Rung 62: G3_BIN_ADD_1
// Tambahkan bobot bit yang aktif
  LD %M120                (* G3_BIN_B0 *)
  [ %MW32 := %MW32 + 1 ]  (* ENC_BINARY_G3, ENC_BINARY_G3 *)
  // as ST:
  //   IF G3_BIN_B0 THEN ENC_BINARY_G3 := ENC_BINARY_G3 + 1; END_IF;

// Rung 63: G3_BIN_ADD_2
// Tambahkan bobot bit yang aktif
  LD %M121                (* G3_BIN_B1 *)
  [ %MW32 := %MW32 + 2 ]  (* ENC_BINARY_G3, ENC_BINARY_G3 *)
  // as ST:
  //   IF G3_BIN_B1 THEN ENC_BINARY_G3 := ENC_BINARY_G3 + 2; END_IF;

// Rung 64: G3_BIN_ADD_4
// Tambahkan bobot bit yang aktif
  LD %M122                (* G3_BIN_B2 *)
  [ %MW32 := %MW32 + 4 ]  (* ENC_BINARY_G3, ENC_BINARY_G3 *)
  // as ST:
  //   IF G3_BIN_B2 THEN ENC_BINARY_G3 := ENC_BINARY_G3 + 4; END_IF;

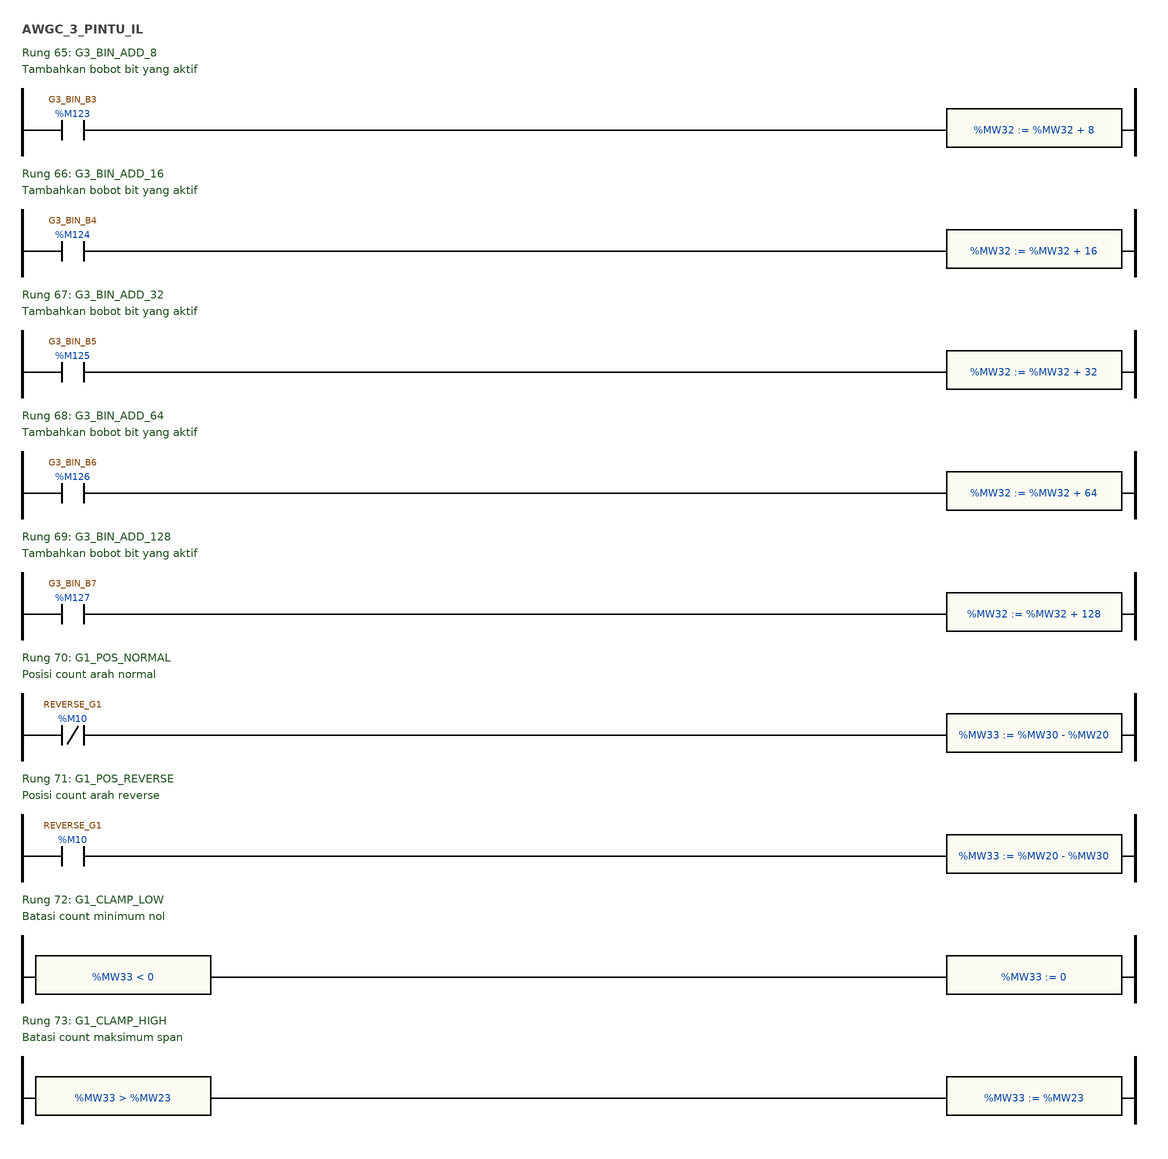

// Rung 65: G3_BIN_ADD_8
// Tambahkan bobot bit yang aktif
  LD %M123                (* G3_BIN_B3 *)
  [ %MW32 := %MW32 + 8 ]  (* ENC_BINARY_G3, ENC_BINARY_G3 *)
  // as ST:
  //   IF G3_BIN_B3 THEN ENC_BINARY_G3 := ENC_BINARY_G3 + 8; END_IF;

// Rung 66: G3_BIN_ADD_16
// Tambahkan bobot bit yang aktif
  LD %M124                (* G3_BIN_B4 *)
  [ %MW32 := %MW32 + 16 ] (* ENC_BINARY_G3, ENC_BINARY_G3 *)
  // as ST:
  //   IF G3_BIN_B4 THEN ENC_BINARY_G3 := ENC_BINARY_G3 + 16; END_IF;

// Rung 67: G3_BIN_ADD_32
// Tambahkan bobot bit yang aktif
  LD %M125                (* G3_BIN_B5 *)
  [ %MW32 := %MW32 + 32 ] (* ENC_BINARY_G3, ENC_BINARY_G3 *)
  // as ST:
  //   IF G3_BIN_B5 THEN ENC_BINARY_G3 := ENC_BINARY_G3 + 32; END_IF;

// Rung 68: G3_BIN_ADD_64
// Tambahkan bobot bit yang aktif
  LD %M126                (* G3_BIN_B6 *)
  [ %MW32 := %MW32 + 64 ] (* ENC_BINARY_G3, ENC_BINARY_G3 *)
  // as ST:
  //   IF G3_BIN_B6 THEN ENC_BINARY_G3 := ENC_BINARY_G3 + 64; END_IF;

// Rung 69: G3_BIN_ADD_128
// Tambahkan bobot bit yang aktif
  LD %M127                (* G3_BIN_B7 *)
  [ %MW32 := %MW32 + 128 ](* ENC_BINARY_G3, ENC_BINARY_G3 *)
  // as ST:
  //   IF G3_BIN_B7 THEN ENC_BINARY_G3 := ENC_BINARY_G3 + 128; END_IF;

// Rung 70: G1_POS_NORMAL
// Posisi count arah normal
  LDN %M10                (* REVERSE_G1 *)
  [ %MW33 := %MW30 - %MW20 ](* POS_COUNT_G1, ENC_BINARY_G1, ENC_ZERO_G1 *)
  // as ST:
  //   IF NOT REVERSE_G1 THEN POS_COUNT_G1 := ENC_BINARY_G1 - ENC_ZERO_G1; END_IF;

// Rung 71: G1_POS_REVERSE
// Posisi count arah reverse
  LD %M10                 (* REVERSE_G1 *)
  [ %MW33 := %MW20 - %MW30 ](* POS_COUNT_G1, ENC_ZERO_G1, ENC_BINARY_G1 *)
  // as ST:
  //   IF REVERSE_G1 THEN POS_COUNT_G1 := ENC_ZERO_G1 - ENC_BINARY_G1; END_IF;

// Rung 72: G1_CLAMP_LOW
// Batasi count minimum nol
  LD [ %MW33 < 0 ]        (* POS_COUNT_G1 *)
  [ %MW33 := 0 ]          (* POS_COUNT_G1 *)
  // as ST:
  //   IF POS_COUNT_G1 < 0 THEN POS_COUNT_G1 := 0; END_IF;

// Rung 73: G1_CLAMP_HIGH
// Batasi count maksimum span
  LD [ %MW33 > %MW23 ]    (* POS_COUNT_G1, ENC_SPAN_G1 *)
  [ %MW33 := %MW23 ]      (* POS_COUNT_G1, ENC_SPAN_G1 *)
  // as ST:
  //   IF POS_COUNT_G1 > ENC_SPAN_G1 THEN POS_COUNT_G1 := ENC_SPAN_G1; END_IF;

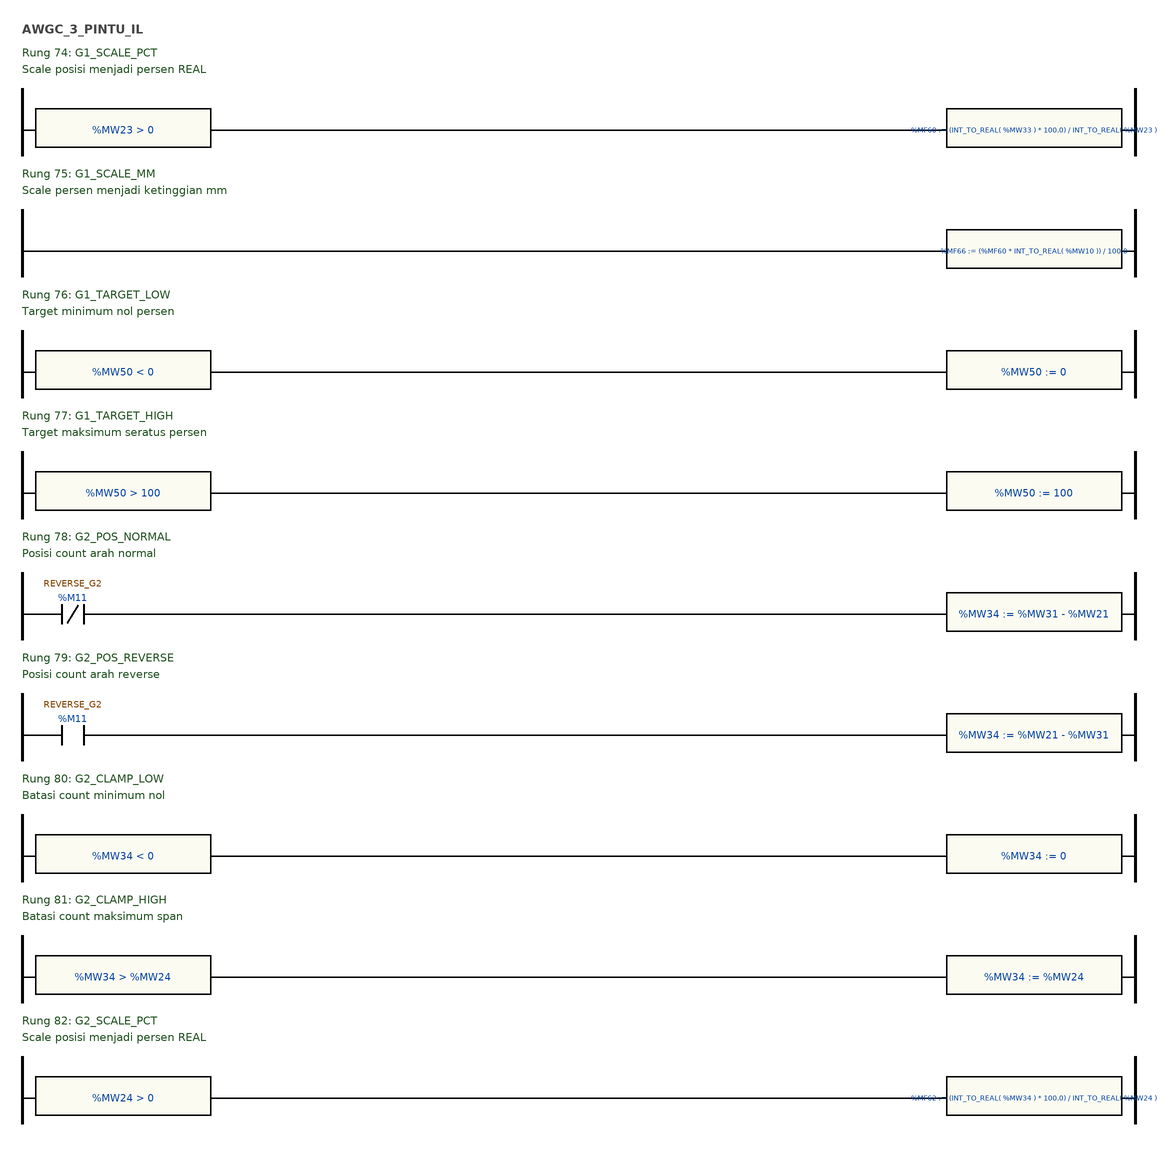

// Rung 74: G1_SCALE_PCT
// Scale posisi menjadi persen REAL
  LD [ %MW23 > 0 ]        (* ENC_SPAN_G1 *)
  [ %MF60 := ( INT_TO_REAL ( %MW33 ) * 100.0 ) / INT_TO_REAL ( %MW23 ) ](* POSITION_G1_PCT, POS_COUNT_G1, ENC_SPAN_G1 *)
  // as ST:
  //   IF ENC_SPAN_G1 > 0 THEN POSITION_G1_PCT := ( INT_TO_REAL ( POS_COUNT_G1 ) * 100.0 ) / INT_TO_REAL ( ENC_SPAN_G1 ); END_IF;

// Rung 75: G1_SCALE_MM
// Scale persen menjadi ketinggian mm
  LD 1
  [ %MF66 := ( %MF60 * INT_TO_REAL ( %MW10 ) ) / 100.0 ](* POSITION_G1_MM, POSITION_G1_PCT, MAX_HEIGHT_G1_MM *)
  // as ST:
  //   POSITION_G1_MM := ( POSITION_G1_PCT * INT_TO_REAL ( MAX_HEIGHT_G1_MM ) ) / 100.0;

// Rung 76: G1_TARGET_LOW
// Target minimum nol persen
  LD [ %MW50 < 0 ]        (* TARGET_PCT_G1 *)
  [ %MW50 := 0 ]          (* TARGET_PCT_G1 *)
  // as ST:
  //   IF TARGET_PCT_G1 < 0 THEN TARGET_PCT_G1 := 0; END_IF;

// Rung 77: G1_TARGET_HIGH
// Target maksimum seratus persen
  LD [ %MW50 > 100 ]      (* TARGET_PCT_G1 *)
  [ %MW50 := 100 ]        (* TARGET_PCT_G1 *)
  // as ST:
  //   IF TARGET_PCT_G1 > 100 THEN TARGET_PCT_G1 := 100; END_IF;

// Rung 78: G2_POS_NORMAL
// Posisi count arah normal
  LDN %M11                (* REVERSE_G2 *)
  [ %MW34 := %MW31 - %MW21 ](* POS_COUNT_G2, ENC_BINARY_G2, ENC_ZERO_G2 *)
  // as ST:
  //   IF NOT REVERSE_G2 THEN POS_COUNT_G2 := ENC_BINARY_G2 - ENC_ZERO_G2; END_IF;

// Rung 79: G2_POS_REVERSE
// Posisi count arah reverse
  LD %M11                 (* REVERSE_G2 *)
  [ %MW34 := %MW21 - %MW31 ](* POS_COUNT_G2, ENC_ZERO_G2, ENC_BINARY_G2 *)
  // as ST:
  //   IF REVERSE_G2 THEN POS_COUNT_G2 := ENC_ZERO_G2 - ENC_BINARY_G2; END_IF;

// Rung 80: G2_CLAMP_LOW
// Batasi count minimum nol
  LD [ %MW34 < 0 ]        (* POS_COUNT_G2 *)
  [ %MW34 := 0 ]          (* POS_COUNT_G2 *)
  // as ST:
  //   IF POS_COUNT_G2 < 0 THEN POS_COUNT_G2 := 0; END_IF;

// Rung 81: G2_CLAMP_HIGH
// Batasi count maksimum span
  LD [ %MW34 > %MW24 ]    (* POS_COUNT_G2, ENC_SPAN_G2 *)
  [ %MW34 := %MW24 ]      (* POS_COUNT_G2, ENC_SPAN_G2 *)
  // as ST:
  //   IF POS_COUNT_G2 > ENC_SPAN_G2 THEN POS_COUNT_G2 := ENC_SPAN_G2; END_IF;

// Rung 82: G2_SCALE_PCT
// Scale posisi menjadi persen REAL
  LD [ %MW24 > 0 ]        (* ENC_SPAN_G2 *)
  [ %MF62 := ( INT_TO_REAL ( %MW34 ) * 100.0 ) / INT_TO_REAL ( %MW24 ) ](* POSITION_G2_PCT, POS_COUNT_G2, ENC_SPAN_G2 *)
  // as ST:
  //   IF ENC_SPAN_G2 > 0 THEN POSITION_G2_PCT := ( INT_TO_REAL ( POS_COUNT_G2 ) * 100.0 ) / INT_TO_REAL ( ENC_SPAN_G2 ); END_IF;

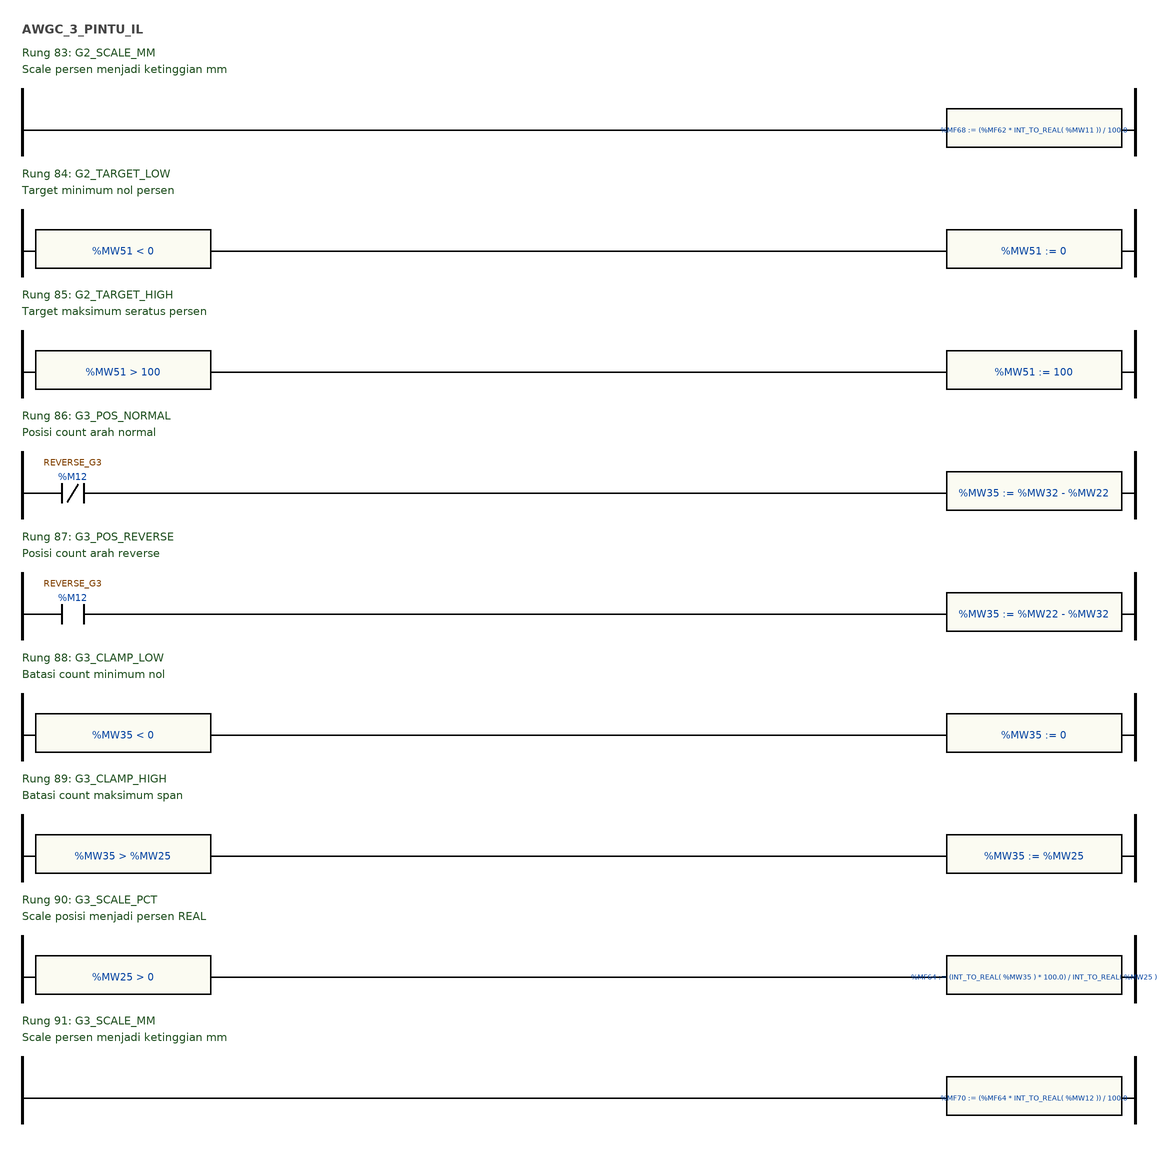

// Rung 83: G2_SCALE_MM
// Scale persen menjadi ketinggian mm
  LD 1
  [ %MF68 := ( %MF62 * INT_TO_REAL ( %MW11 ) ) / 100.0 ](* POSITION_G2_MM, POSITION_G2_PCT, MAX_HEIGHT_G2_MM *)
  // as ST:
  //   POSITION_G2_MM := ( POSITION_G2_PCT * INT_TO_REAL ( MAX_HEIGHT_G2_MM ) ) / 100.0;

// Rung 84: G2_TARGET_LOW
// Target minimum nol persen
  LD [ %MW51 < 0 ]        (* TARGET_PCT_G2 *)
  [ %MW51 := 0 ]          (* TARGET_PCT_G2 *)
  // as ST:
  //   IF TARGET_PCT_G2 < 0 THEN TARGET_PCT_G2 := 0; END_IF;

// Rung 85: G2_TARGET_HIGH
// Target maksimum seratus persen
  LD [ %MW51 > 100 ]      (* TARGET_PCT_G2 *)
  [ %MW51 := 100 ]        (* TARGET_PCT_G2 *)
  // as ST:
  //   IF TARGET_PCT_G2 > 100 THEN TARGET_PCT_G2 := 100; END_IF;

// Rung 86: G3_POS_NORMAL
// Posisi count arah normal
  LDN %M12                (* REVERSE_G3 *)
  [ %MW35 := %MW32 - %MW22 ](* POS_COUNT_G3, ENC_BINARY_G3, ENC_ZERO_G3 *)
  // as ST:
  //   IF NOT REVERSE_G3 THEN POS_COUNT_G3 := ENC_BINARY_G3 - ENC_ZERO_G3; END_IF;

// Rung 87: G3_POS_REVERSE
// Posisi count arah reverse
  LD %M12                 (* REVERSE_G3 *)
  [ %MW35 := %MW22 - %MW32 ](* POS_COUNT_G3, ENC_ZERO_G3, ENC_BINARY_G3 *)
  // as ST:
  //   IF REVERSE_G3 THEN POS_COUNT_G3 := ENC_ZERO_G3 - ENC_BINARY_G3; END_IF;

// Rung 88: G3_CLAMP_LOW
// Batasi count minimum nol
  LD [ %MW35 < 0 ]        (* POS_COUNT_G3 *)
  [ %MW35 := 0 ]          (* POS_COUNT_G3 *)
  // as ST:
  //   IF POS_COUNT_G3 < 0 THEN POS_COUNT_G3 := 0; END_IF;

// Rung 89: G3_CLAMP_HIGH
// Batasi count maksimum span
  LD [ %MW35 > %MW25 ]    (* POS_COUNT_G3, ENC_SPAN_G3 *)
  [ %MW35 := %MW25 ]      (* POS_COUNT_G3, ENC_SPAN_G3 *)
  // as ST:
  //   IF POS_COUNT_G3 > ENC_SPAN_G3 THEN POS_COUNT_G3 := ENC_SPAN_G3; END_IF;

// Rung 90: G3_SCALE_PCT
// Scale posisi menjadi persen REAL
  LD [ %MW25 > 0 ]        (* ENC_SPAN_G3 *)
  [ %MF64 := ( INT_TO_REAL ( %MW35 ) * 100.0 ) / INT_TO_REAL ( %MW25 ) ](* POSITION_G3_PCT, POS_COUNT_G3, ENC_SPAN_G3 *)
  // as ST:
  //   IF ENC_SPAN_G3 > 0 THEN POSITION_G3_PCT := ( INT_TO_REAL ( POS_COUNT_G3 ) * 100.0 ) / INT_TO_REAL ( ENC_SPAN_G3 ); END_IF;

// Rung 91: G3_SCALE_MM
// Scale persen menjadi ketinggian mm
  LD 1
  [ %MF70 := ( %MF64 * INT_TO_REAL ( %MW12 ) ) / 100.0 ](* POSITION_G3_MM, POSITION_G3_PCT, MAX_HEIGHT_G3_MM *)
  // as ST:
  //   POSITION_G3_MM := ( POSITION_G3_PCT * INT_TO_REAL ( MAX_HEIGHT_G3_MM ) ) / 100.0;

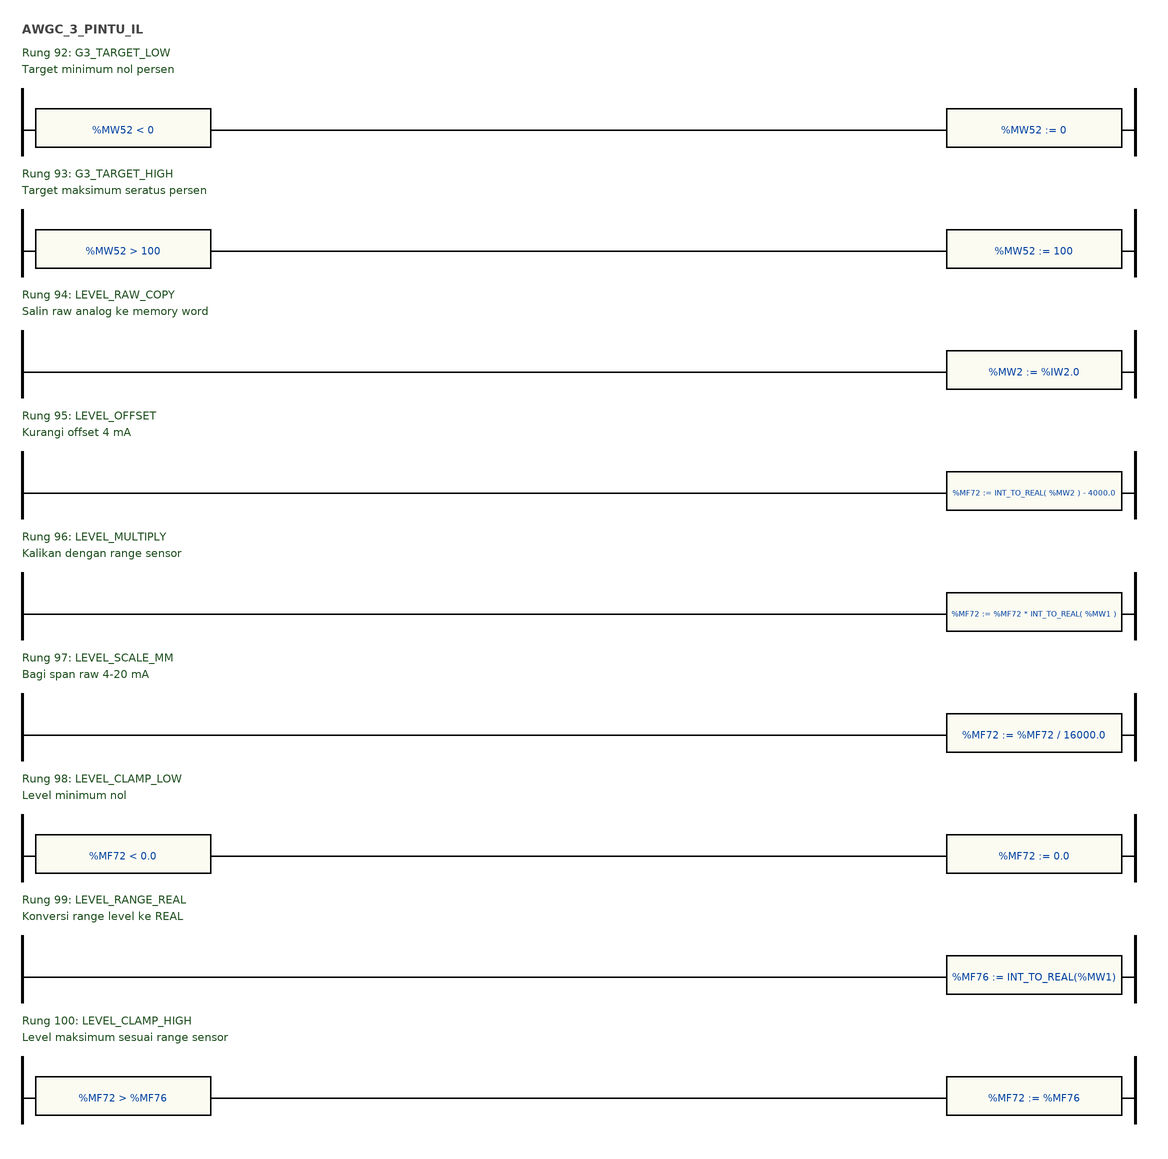

// Rung 92: G3_TARGET_LOW
// Target minimum nol persen
  LD [ %MW52 < 0 ]        (* TARGET_PCT_G3 *)
  [ %MW52 := 0 ]          (* TARGET_PCT_G3 *)
  // as ST:
  //   IF TARGET_PCT_G3 < 0 THEN TARGET_PCT_G3 := 0; END_IF;

// Rung 93: G3_TARGET_HIGH
// Target maksimum seratus persen
  LD [ %MW52 > 100 ]      (* TARGET_PCT_G3 *)
  [ %MW52 := 100 ]        (* TARGET_PCT_G3 *)
  // as ST:
  //   IF TARGET_PCT_G3 > 100 THEN TARGET_PCT_G3 := 100; END_IF;

// Rung 94: LEVEL_RAW_COPY
// Salin raw analog ke memory word
  LD 1
  [ %MW2 := %IW2.0 ]      (* LEVEL_RAW_COPY, LEVEL_RAW *)
  // as ST:
  //   LEVEL_RAW_COPY := LEVEL_RAW;

// Rung 95: LEVEL_OFFSET
// Kurangi offset 4 mA
  LD 1
  [ %MF72 := INT_TO_REAL ( %MW2 ) - 4000.0 ](* WATER_LEVEL_MM, LEVEL_RAW_COPY *)
  // as ST:
  //   WATER_LEVEL_MM := INT_TO_REAL ( LEVEL_RAW_COPY ) - 4000.0;

// Rung 96: LEVEL_MULTIPLY
// Kalikan dengan range sensor
  LD 1
  [ %MF72 := %MF72 * INT_TO_REAL ( %MW1 ) ](* WATER_LEVEL_MM, WATER_LEVEL_MM, WATER_RANGE_MM *)
  // as ST:
  //   WATER_LEVEL_MM := WATER_LEVEL_MM * INT_TO_REAL ( WATER_RANGE_MM );

// Rung 97: LEVEL_SCALE_MM
// Bagi span raw 4-20 mA
  LD 1
  [ %MF72 := %MF72 / 16000.0 ](* WATER_LEVEL_MM, WATER_LEVEL_MM *)
  // as ST:
  //   WATER_LEVEL_MM := WATER_LEVEL_MM / 16000.0;

// Rung 98: LEVEL_CLAMP_LOW
// Level minimum nol
  LD [ %MF72 < 0.0 ]      (* WATER_LEVEL_MM *)
  [ %MF72 := 0.0 ]        (* WATER_LEVEL_MM *)
  // as ST:
  //   IF WATER_LEVEL_MM < 0.0 THEN WATER_LEVEL_MM := 0.0; END_IF;

// Rung 99: LEVEL_RANGE_REAL
// Konversi range level ke REAL
  LD 1
  [ %MF76 := INT_TO_REAL ( %MW1 ) ](* WATER_RANGE_REAL, WATER_RANGE_MM *)
  // as ST:
  //   WATER_RANGE_REAL := INT_TO_REAL ( WATER_RANGE_MM );

// Rung 100: LEVEL_CLAMP_HIGH
// Level maksimum sesuai range sensor
  LD [ %MF72 > %MF76 ]    (* WATER_LEVEL_MM, WATER_RANGE_REAL *)
  [ %MF72 := %MF76 ]      (* WATER_LEVEL_MM, WATER_RANGE_REAL *)
  // as ST:
  //   IF WATER_LEVEL_MM > WATER_RANGE_REAL THEN WATER_LEVEL_MM := WATER_RANGE_REAL; END_IF;

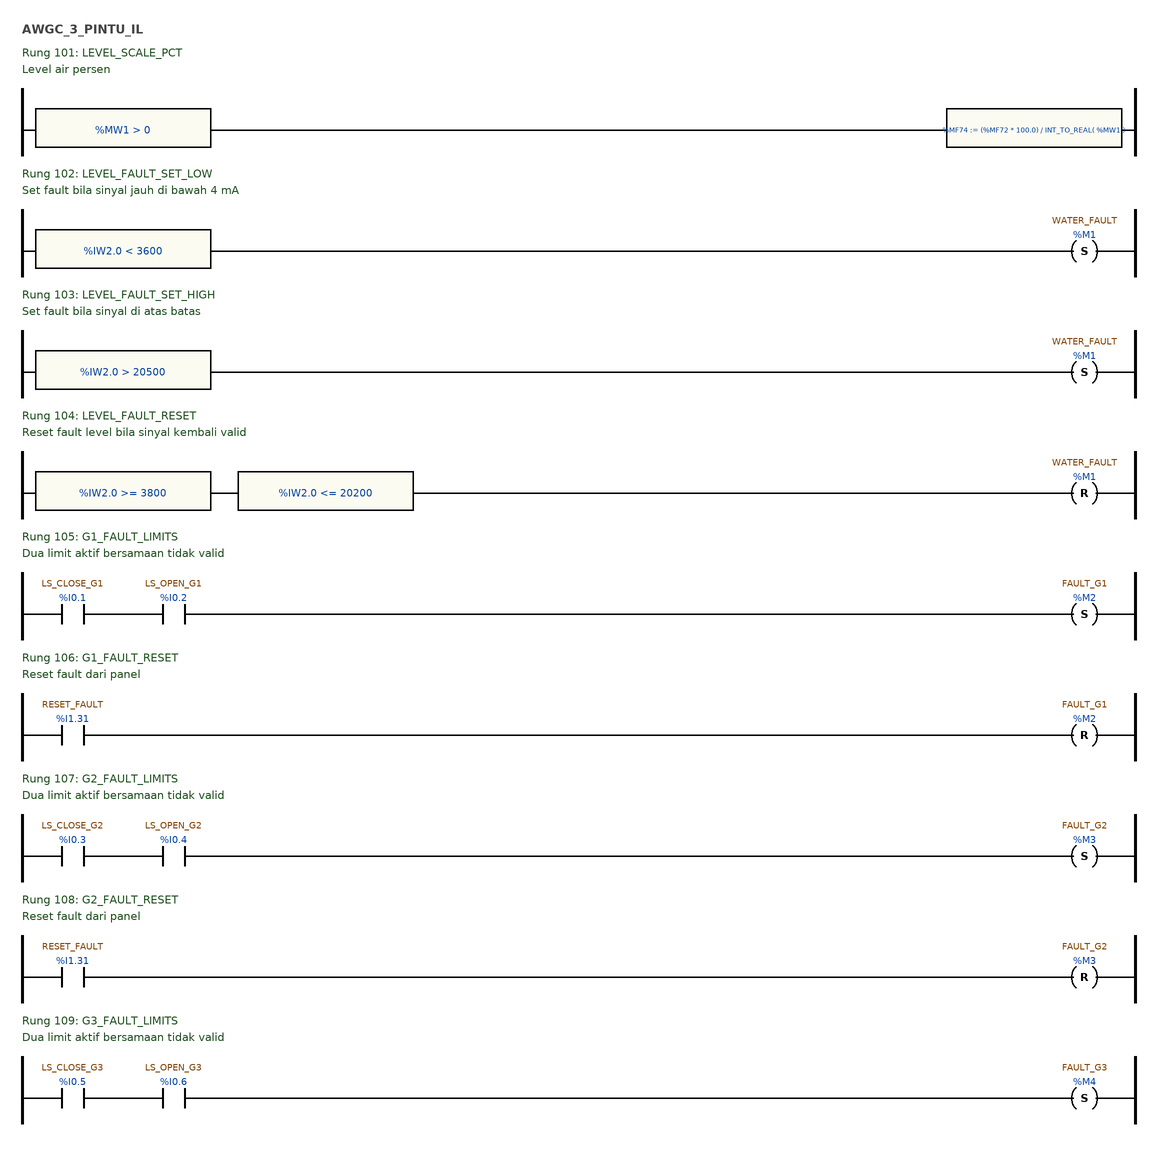

// Rung 101: LEVEL_SCALE_PCT
// Level air persen
  LD [ %MW1 > 0 ]         (* WATER_RANGE_MM *)
  [ %MF74 := ( %MF72 * 100.0 ) / INT_TO_REAL ( %MW1 ) ](* WATER_LEVEL_PCT, WATER_LEVEL_MM, WATER_RANGE_MM *)
  // as ST:
  //   IF WATER_RANGE_MM > 0 THEN WATER_LEVEL_PCT := ( WATER_LEVEL_MM * 100.0 ) / INT_TO_REAL ( WATER_RANGE_MM ); END_IF;

// Rung 102: LEVEL_FAULT_SET_LOW
// Set fault bila sinyal jauh di bawah 4 mA
  LD [ %IW2.0 < 3600 ]    (* LEVEL_RAW *)
  S %M1                   (* WATER_FAULT *)
  // as ST:
  //   IF LEVEL_RAW < 3600 THEN WATER_FAULT := TRUE; END_IF;

// Rung 103: LEVEL_FAULT_SET_HIGH
// Set fault bila sinyal di atas batas
  LD [ %IW2.0 > 20500 ]   (* LEVEL_RAW *)
  S %M1                   (* WATER_FAULT *)
  // as ST:
  //   IF LEVEL_RAW > 20500 THEN WATER_FAULT := TRUE; END_IF;

// Rung 104: LEVEL_FAULT_RESET
// Reset fault level bila sinyal kembali valid
  LD [ %IW2.0 >= 3800 ]   (* LEVEL_RAW *)
  AND [ %IW2.0 <= 20200 ] (* LEVEL_RAW *)
  R %M1                   (* WATER_FAULT *)
  // as ST:
  //   IF LEVEL_RAW >= 3800 AND LEVEL_RAW <= 20200 THEN WATER_FAULT := FALSE; END_IF;

// Rung 105: G1_FAULT_LIMITS
// Dua limit aktif bersamaan tidak valid
  LD %I0.1                (* LS_CLOSE_G1 *)
  AND %I0.2               (* LS_OPEN_G1 *)
  S %M2                   (* FAULT_G1 *)
  // as ST:
  //   IF LS_CLOSE_G1 AND LS_OPEN_G1 THEN FAULT_G1 := TRUE; END_IF;

// Rung 106: G1_FAULT_RESET
// Reset fault dari panel
  LD %I1.31               (* RESET_FAULT *)
  R %M2                   (* FAULT_G1 *)
  // as ST:
  //   IF RESET_FAULT THEN FAULT_G1 := FALSE; END_IF;

// Rung 107: G2_FAULT_LIMITS
// Dua limit aktif bersamaan tidak valid
  LD %I0.3                (* LS_CLOSE_G2 *)
  AND %I0.4               (* LS_OPEN_G2 *)
  S %M3                   (* FAULT_G2 *)
  // as ST:
  //   IF LS_CLOSE_G2 AND LS_OPEN_G2 THEN FAULT_G2 := TRUE; END_IF;

// Rung 108: G2_FAULT_RESET
// Reset fault dari panel
  LD %I1.31               (* RESET_FAULT *)
  R %M3                   (* FAULT_G2 *)
  // as ST:
  //   IF RESET_FAULT THEN FAULT_G2 := FALSE; END_IF;

// Rung 109: G3_FAULT_LIMITS
// Dua limit aktif bersamaan tidak valid
  LD %I0.5                (* LS_CLOSE_G3 *)
  AND %I0.6               (* LS_OPEN_G3 *)
  S %M4                   (* FAULT_G3 *)
  // as ST:
  //   IF LS_CLOSE_G3 AND LS_OPEN_G3 THEN FAULT_G3 := TRUE; END_IF;

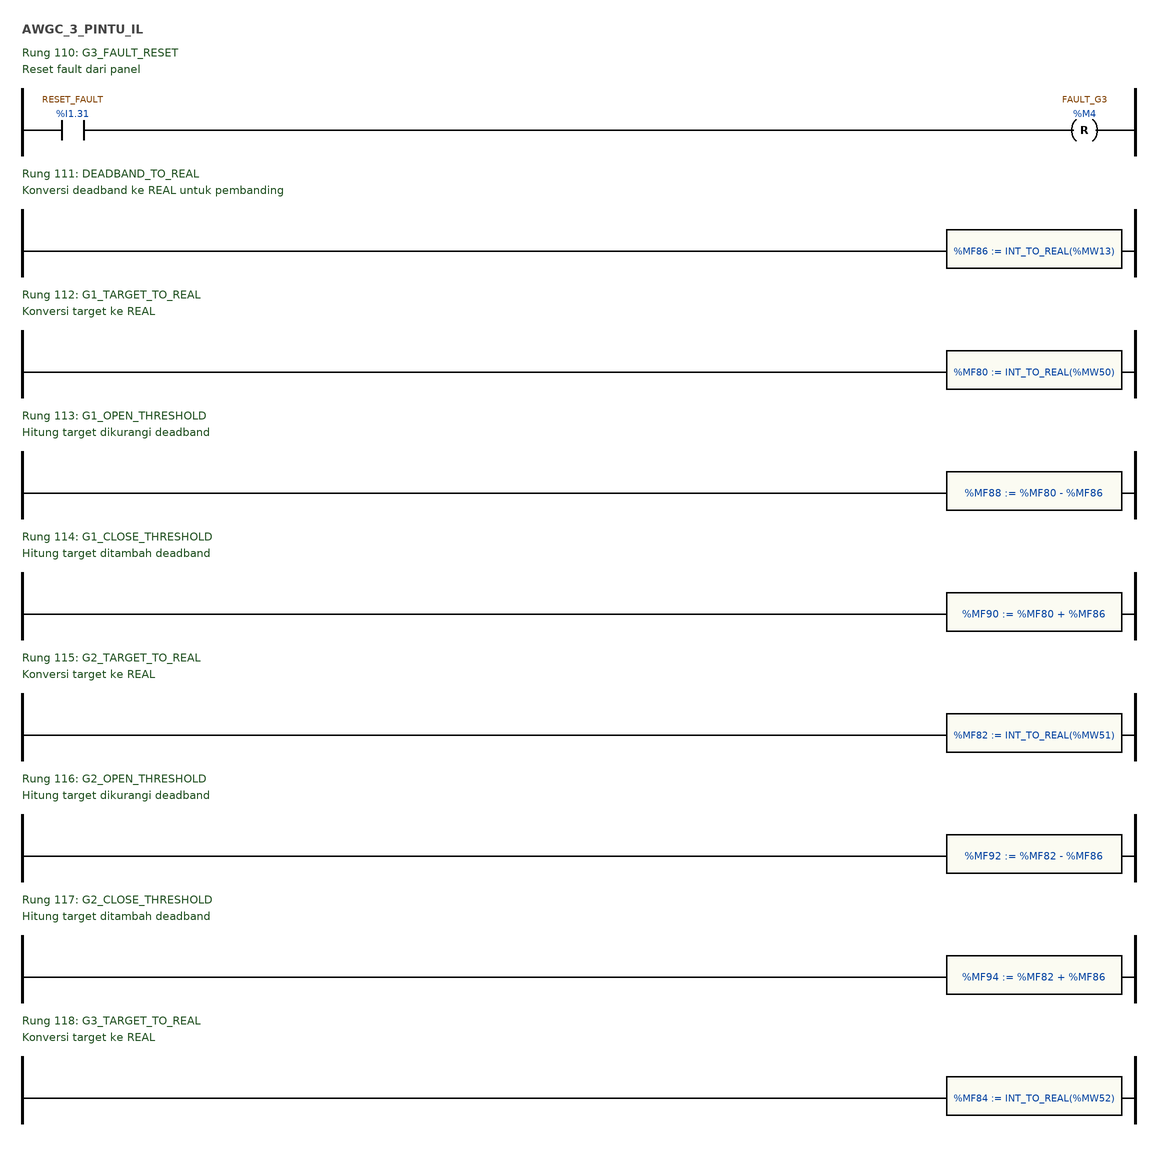

// Rung 110: G3_FAULT_RESET
// Reset fault dari panel
  LD %I1.31               (* RESET_FAULT *)
  R %M4                   (* FAULT_G3 *)
  // as ST:
  //   IF RESET_FAULT THEN FAULT_G3 := FALSE; END_IF;

// Rung 111: DEADBAND_TO_REAL
// Konversi deadband ke REAL untuk pembanding
  LD 1
  [ %MF86 := INT_TO_REAL ( %MW13 ) ](* DEADBAND_REAL, DEADBAND_PCT *)
  // as ST:
  //   DEADBAND_REAL := INT_TO_REAL ( DEADBAND_PCT );

// Rung 112: G1_TARGET_TO_REAL
// Konversi target ke REAL
  LD 1
  [ %MF80 := INT_TO_REAL ( %MW50 ) ](* TARGET_G1_REAL, TARGET_PCT_G1 *)
  // as ST:
  //   TARGET_G1_REAL := INT_TO_REAL ( TARGET_PCT_G1 );

// Rung 113: G1_OPEN_THRESHOLD
// Hitung target dikurangi deadband
  LD 1
  [ %MF88 := %MF80 - %MF86 ](* OPEN_THRESHOLD_G1, TARGET_G1_REAL, DEADBAND_REAL *)
  // as ST:
  //   OPEN_THRESHOLD_G1 := TARGET_G1_REAL - DEADBAND_REAL;

// Rung 114: G1_CLOSE_THRESHOLD
// Hitung target ditambah deadband
  LD 1
  [ %MF90 := %MF80 + %MF86 ](* CLOSE_THRESHOLD_G1, TARGET_G1_REAL, DEADBAND_REAL *)
  // as ST:
  //   CLOSE_THRESHOLD_G1 := TARGET_G1_REAL + DEADBAND_REAL;

// Rung 115: G2_TARGET_TO_REAL
// Konversi target ke REAL
  LD 1
  [ %MF82 := INT_TO_REAL ( %MW51 ) ](* TARGET_G2_REAL, TARGET_PCT_G2 *)
  // as ST:
  //   TARGET_G2_REAL := INT_TO_REAL ( TARGET_PCT_G2 );

// Rung 116: G2_OPEN_THRESHOLD
// Hitung target dikurangi deadband
  LD 1
  [ %MF92 := %MF82 - %MF86 ](* OPEN_THRESHOLD_G2, TARGET_G2_REAL, DEADBAND_REAL *)
  // as ST:
  //   OPEN_THRESHOLD_G2 := TARGET_G2_REAL - DEADBAND_REAL;

// Rung 117: G2_CLOSE_THRESHOLD
// Hitung target ditambah deadband
  LD 1
  [ %MF94 := %MF82 + %MF86 ](* CLOSE_THRESHOLD_G2, TARGET_G2_REAL, DEADBAND_REAL *)
  // as ST:
  //   CLOSE_THRESHOLD_G2 := TARGET_G2_REAL + DEADBAND_REAL;

// Rung 118: G3_TARGET_TO_REAL
// Konversi target ke REAL
  LD 1
  [ %MF84 := INT_TO_REAL ( %MW52 ) ](* TARGET_G3_REAL, TARGET_PCT_G3 *)
  // as ST:
  //   TARGET_G3_REAL := INT_TO_REAL ( TARGET_PCT_G3 );

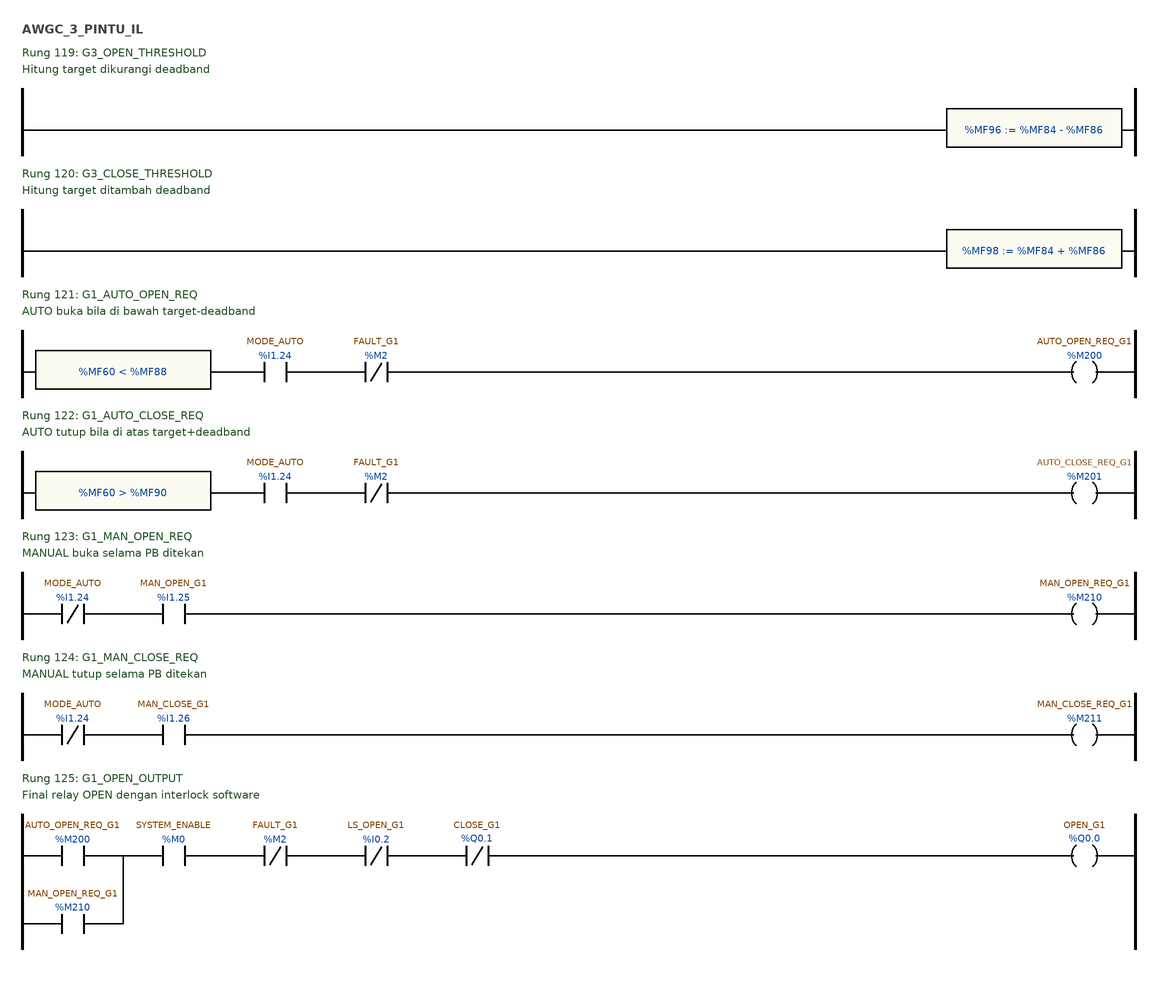

// Rung 119: G3_OPEN_THRESHOLD
// Hitung target dikurangi deadband
  LD 1
  [ %MF96 := %MF84 - %MF86 ](* OPEN_THRESHOLD_G3, TARGET_G3_REAL, DEADBAND_REAL *)
  // as ST:
  //   OPEN_THRESHOLD_G3 := TARGET_G3_REAL - DEADBAND_REAL;

// Rung 120: G3_CLOSE_THRESHOLD
// Hitung target ditambah deadband
  LD 1
  [ %MF98 := %MF84 + %MF86 ](* CLOSE_THRESHOLD_G3, TARGET_G3_REAL, DEADBAND_REAL *)
  // as ST:
  //   CLOSE_THRESHOLD_G3 := TARGET_G3_REAL + DEADBAND_REAL;

// Rung 121: G1_AUTO_OPEN_REQ
// AUTO buka bila di bawah target-deadband
  LD [ %MF60 < %MF88 ]    (* POSITION_G1_PCT, OPEN_THRESHOLD_G1 *)
  AND %I1.24              (* MODE_AUTO *)
  ANDN %M2                (* FAULT_G1 *)
  ST %M200                (* AUTO_OPEN_REQ_G1 *)
  // as ST:
  //   AUTO_OPEN_REQ_G1 := POSITION_G1_PCT < OPEN_THRESHOLD_G1 AND MODE_AUTO AND NOT FAULT_G1;

// Rung 122: G1_AUTO_CLOSE_REQ
// AUTO tutup bila di atas target+deadband
  LD [ %MF60 > %MF90 ]    (* POSITION_G1_PCT, CLOSE_THRESHOLD_G1 *)
  AND %I1.24              (* MODE_AUTO *)
  ANDN %M2                (* FAULT_G1 *)
  ST %M201                (* AUTO_CLOSE_REQ_G1 *)
  // as ST:
  //   AUTO_CLOSE_REQ_G1 := POSITION_G1_PCT > CLOSE_THRESHOLD_G1 AND MODE_AUTO AND NOT FAULT_G1;

// Rung 123: G1_MAN_OPEN_REQ
// MANUAL buka selama PB ditekan
  LDN %I1.24              (* MODE_AUTO *)
  AND %I1.25              (* MAN_OPEN_G1 *)
  ST %M210                (* MAN_OPEN_REQ_G1 *)
  // as ST:
  //   MAN_OPEN_REQ_G1 := NOT MODE_AUTO AND MAN_OPEN_G1;

// Rung 124: G1_MAN_CLOSE_REQ
// MANUAL tutup selama PB ditekan
  LDN %I1.24              (* MODE_AUTO *)
  AND %I1.26              (* MAN_CLOSE_G1 *)
  ST %M211                (* MAN_CLOSE_REQ_G1 *)
  // as ST:
  //   MAN_CLOSE_REQ_G1 := NOT MODE_AUTO AND MAN_CLOSE_G1;

// Rung 125: G1_OPEN_OUTPUT
// Final relay OPEN dengan interlock software
  LD %M200                (* AUTO_OPEN_REQ_G1 *)
  OR %M210                (* MAN_OPEN_REQ_G1 *)
  AND %M0                 (* SYSTEM_ENABLE *)
  ANDN %M2                (* FAULT_G1 *)
  ANDN %I0.2              (* LS_OPEN_G1 *)
  ANDN %Q0.1              (* CLOSE_G1 *)
  ST %Q0.0                (* OPEN_G1 *)
  // as ST:
  //   OPEN_G1 := (AUTO_OPEN_REQ_G1 OR MAN_OPEN_REQ_G1) AND SYSTEM_ENABLE AND NOT FAULT_G1 AND NOT LS_OPEN_G1 AND NOT CLOSE_G1;

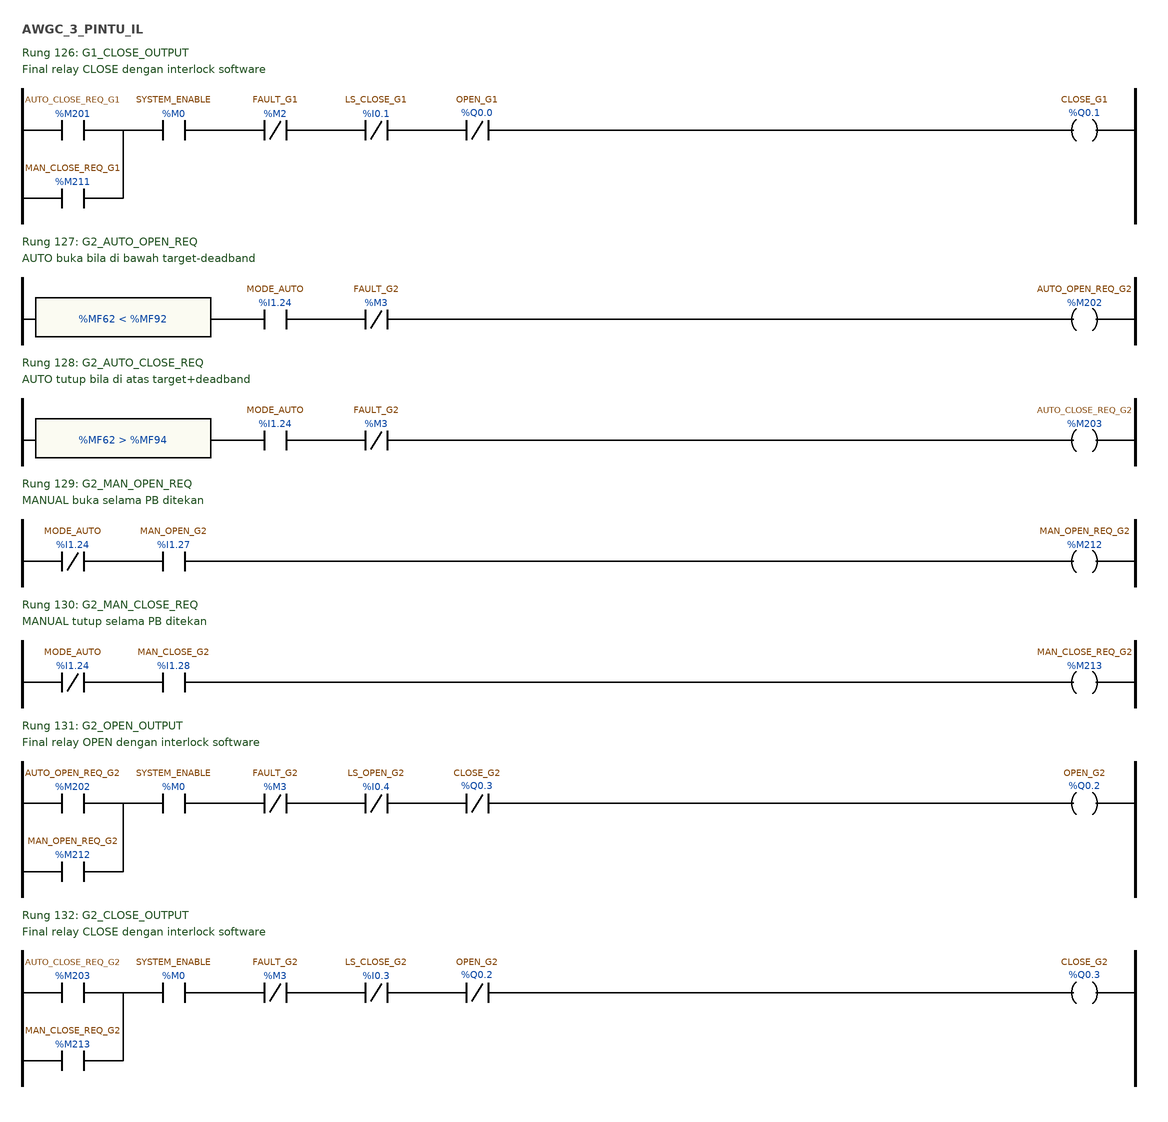

// Rung 126: G1_CLOSE_OUTPUT
// Final relay CLOSE dengan interlock software
  LD %M201                (* AUTO_CLOSE_REQ_G1 *)
  OR %M211                (* MAN_CLOSE_REQ_G1 *)
  AND %M0                 (* SYSTEM_ENABLE *)
  ANDN %M2                (* FAULT_G1 *)
  ANDN %I0.1              (* LS_CLOSE_G1 *)
  ANDN %Q0.0              (* OPEN_G1 *)
  ST %Q0.1                (* CLOSE_G1 *)
  // as ST:
  //   CLOSE_G1 := (AUTO_CLOSE_REQ_G1 OR MAN_CLOSE_REQ_G1) AND SYSTEM_ENABLE AND NOT FAULT_G1 AND NOT LS_CLOSE_G1 AND NOT OPEN_G1;

// Rung 127: G2_AUTO_OPEN_REQ
// AUTO buka bila di bawah target-deadband
  LD [ %MF62 < %MF92 ]    (* POSITION_G2_PCT, OPEN_THRESHOLD_G2 *)
  AND %I1.24              (* MODE_AUTO *)
  ANDN %M3                (* FAULT_G2 *)
  ST %M202                (* AUTO_OPEN_REQ_G2 *)
  // as ST:
  //   AUTO_OPEN_REQ_G2 := POSITION_G2_PCT < OPEN_THRESHOLD_G2 AND MODE_AUTO AND NOT FAULT_G2;

// Rung 128: G2_AUTO_CLOSE_REQ
// AUTO tutup bila di atas target+deadband
  LD [ %MF62 > %MF94 ]    (* POSITION_G2_PCT, CLOSE_THRESHOLD_G2 *)
  AND %I1.24              (* MODE_AUTO *)
  ANDN %M3                (* FAULT_G2 *)
  ST %M203                (* AUTO_CLOSE_REQ_G2 *)
  // as ST:
  //   AUTO_CLOSE_REQ_G2 := POSITION_G2_PCT > CLOSE_THRESHOLD_G2 AND MODE_AUTO AND NOT FAULT_G2;

// Rung 129: G2_MAN_OPEN_REQ
// MANUAL buka selama PB ditekan
  LDN %I1.24              (* MODE_AUTO *)
  AND %I1.27              (* MAN_OPEN_G2 *)
  ST %M212                (* MAN_OPEN_REQ_G2 *)
  // as ST:
  //   MAN_OPEN_REQ_G2 := NOT MODE_AUTO AND MAN_OPEN_G2;

// Rung 130: G2_MAN_CLOSE_REQ
// MANUAL tutup selama PB ditekan
  LDN %I1.24              (* MODE_AUTO *)
  AND %I1.28              (* MAN_CLOSE_G2 *)
  ST %M213                (* MAN_CLOSE_REQ_G2 *)
  // as ST:
  //   MAN_CLOSE_REQ_G2 := NOT MODE_AUTO AND MAN_CLOSE_G2;

// Rung 131: G2_OPEN_OUTPUT
// Final relay OPEN dengan interlock software
  LD %M202                (* AUTO_OPEN_REQ_G2 *)
  OR %M212                (* MAN_OPEN_REQ_G2 *)
  AND %M0                 (* SYSTEM_ENABLE *)
  ANDN %M3                (* FAULT_G2 *)
  ANDN %I0.4              (* LS_OPEN_G2 *)
  ANDN %Q0.3              (* CLOSE_G2 *)
  ST %Q0.2                (* OPEN_G2 *)
  // as ST:
  //   OPEN_G2 := (AUTO_OPEN_REQ_G2 OR MAN_OPEN_REQ_G2) AND SYSTEM_ENABLE AND NOT FAULT_G2 AND NOT LS_OPEN_G2 AND NOT CLOSE_G2;

// Rung 132: G2_CLOSE_OUTPUT
// Final relay CLOSE dengan interlock software
  LD %M203                (* AUTO_CLOSE_REQ_G2 *)
  OR %M213                (* MAN_CLOSE_REQ_G2 *)
  AND %M0                 (* SYSTEM_ENABLE *)
  ANDN %M3                (* FAULT_G2 *)
  ANDN %I0.3              (* LS_CLOSE_G2 *)
  ANDN %Q0.2              (* OPEN_G2 *)
  ST %Q0.3                (* CLOSE_G2 *)
  // as ST:
  //   CLOSE_G2 := (AUTO_CLOSE_REQ_G2 OR MAN_CLOSE_REQ_G2) AND SYSTEM_ENABLE AND NOT FAULT_G2 AND NOT LS_CLOSE_G2 AND NOT OPEN_G2;

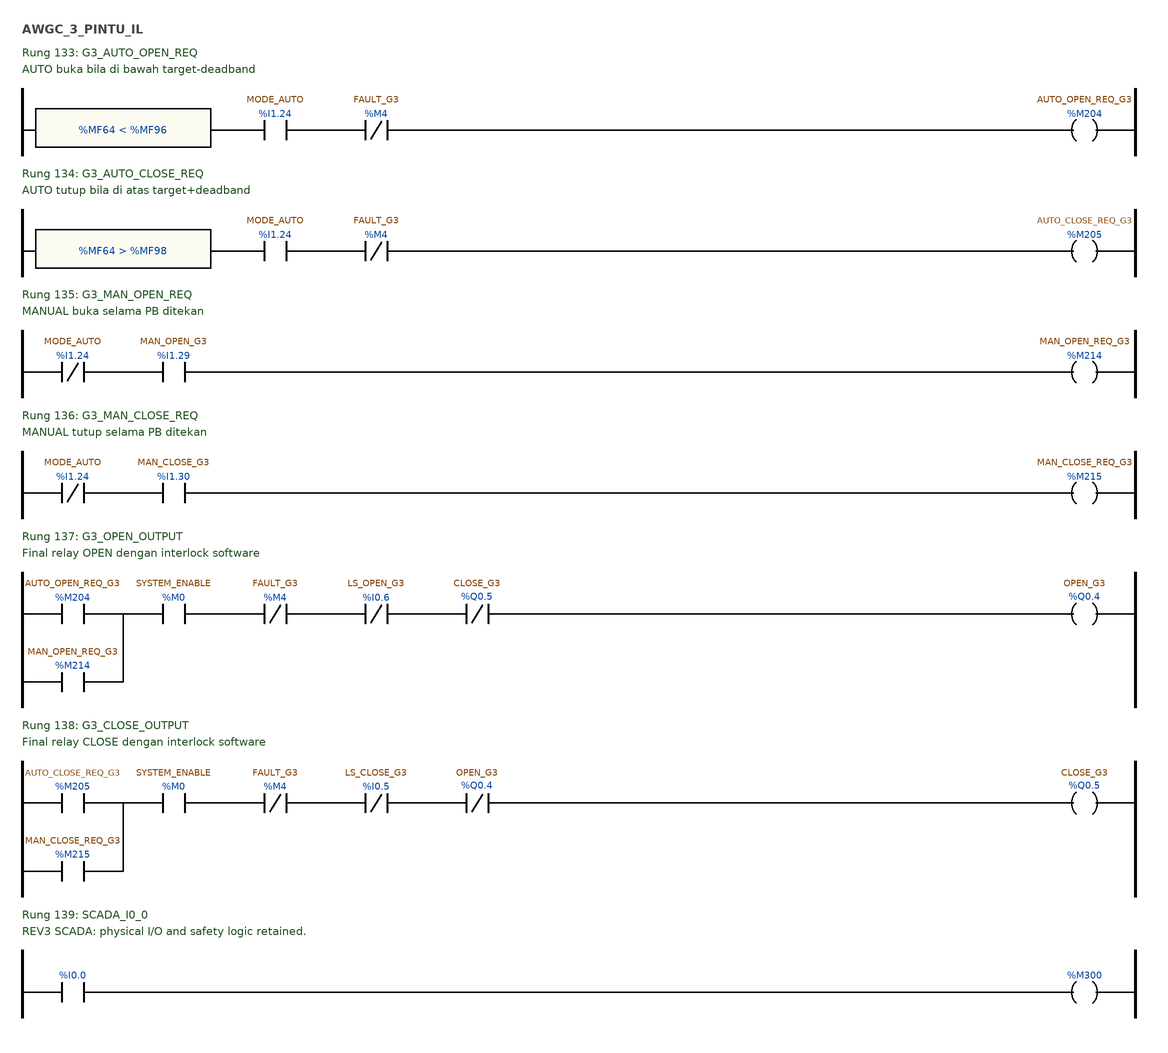

// Rung 133: G3_AUTO_OPEN_REQ
// AUTO buka bila di bawah target-deadband
  LD [ %MF64 < %MF96 ]    (* POSITION_G3_PCT, OPEN_THRESHOLD_G3 *)
  AND %I1.24              (* MODE_AUTO *)
  ANDN %M4                (* FAULT_G3 *)
  ST %M204                (* AUTO_OPEN_REQ_G3 *)
  // as ST:
  //   AUTO_OPEN_REQ_G3 := POSITION_G3_PCT < OPEN_THRESHOLD_G3 AND MODE_AUTO AND NOT FAULT_G3;

// Rung 134: G3_AUTO_CLOSE_REQ
// AUTO tutup bila di atas target+deadband
  LD [ %MF64 > %MF98 ]    (* POSITION_G3_PCT, CLOSE_THRESHOLD_G3 *)
  AND %I1.24              (* MODE_AUTO *)
  ANDN %M4                (* FAULT_G3 *)
  ST %M205                (* AUTO_CLOSE_REQ_G3 *)
  // as ST:
  //   AUTO_CLOSE_REQ_G3 := POSITION_G3_PCT > CLOSE_THRESHOLD_G3 AND MODE_AUTO AND NOT FAULT_G3;

// Rung 135: G3_MAN_OPEN_REQ
// MANUAL buka selama PB ditekan
  LDN %I1.24              (* MODE_AUTO *)
  AND %I1.29              (* MAN_OPEN_G3 *)
  ST %M214                (* MAN_OPEN_REQ_G3 *)
  // as ST:
  //   MAN_OPEN_REQ_G3 := NOT MODE_AUTO AND MAN_OPEN_G3;

// Rung 136: G3_MAN_CLOSE_REQ
// MANUAL tutup selama PB ditekan
  LDN %I1.24              (* MODE_AUTO *)
  AND %I1.30              (* MAN_CLOSE_G3 *)
  ST %M215                (* MAN_CLOSE_REQ_G3 *)
  // as ST:
  //   MAN_CLOSE_REQ_G3 := NOT MODE_AUTO AND MAN_CLOSE_G3;

// Rung 137: G3_OPEN_OUTPUT
// Final relay OPEN dengan interlock software
  LD %M204                (* AUTO_OPEN_REQ_G3 *)
  OR %M214                (* MAN_OPEN_REQ_G3 *)
  AND %M0                 (* SYSTEM_ENABLE *)
  ANDN %M4                (* FAULT_G3 *)
  ANDN %I0.6              (* LS_OPEN_G3 *)
  ANDN %Q0.5              (* CLOSE_G3 *)
  ST %Q0.4                (* OPEN_G3 *)
  // as ST:
  //   OPEN_G3 := (AUTO_OPEN_REQ_G3 OR MAN_OPEN_REQ_G3) AND SYSTEM_ENABLE AND NOT FAULT_G3 AND NOT LS_OPEN_G3 AND NOT CLOSE_G3;

// Rung 138: G3_CLOSE_OUTPUT
// Final relay CLOSE dengan interlock software
  LD %M205                (* AUTO_CLOSE_REQ_G3 *)
  OR %M215                (* MAN_CLOSE_REQ_G3 *)
  AND %M0                 (* SYSTEM_ENABLE *)
  ANDN %M4                (* FAULT_G3 *)
  ANDN %I0.5              (* LS_CLOSE_G3 *)
  ANDN %Q0.4              (* OPEN_G3 *)
  ST %Q0.5                (* CLOSE_G3 *)
  // as ST:
  //   CLOSE_G3 := (AUTO_CLOSE_REQ_G3 OR MAN_CLOSE_REQ_G3) AND SYSTEM_ENABLE AND NOT FAULT_G3 AND NOT LS_CLOSE_G3 AND NOT OPEN_G3;

// Rung 139: SCADA_I0_0
// REV3 SCADA: physical I/O and safety logic retained.
  LD %I0.0                (* SAFETY_OK_IN *)
  ST %M300                (* STATUS_I0_0 *)
  // as ST:
  //   STATUS_I0_0 := SAFETY_OK_IN;

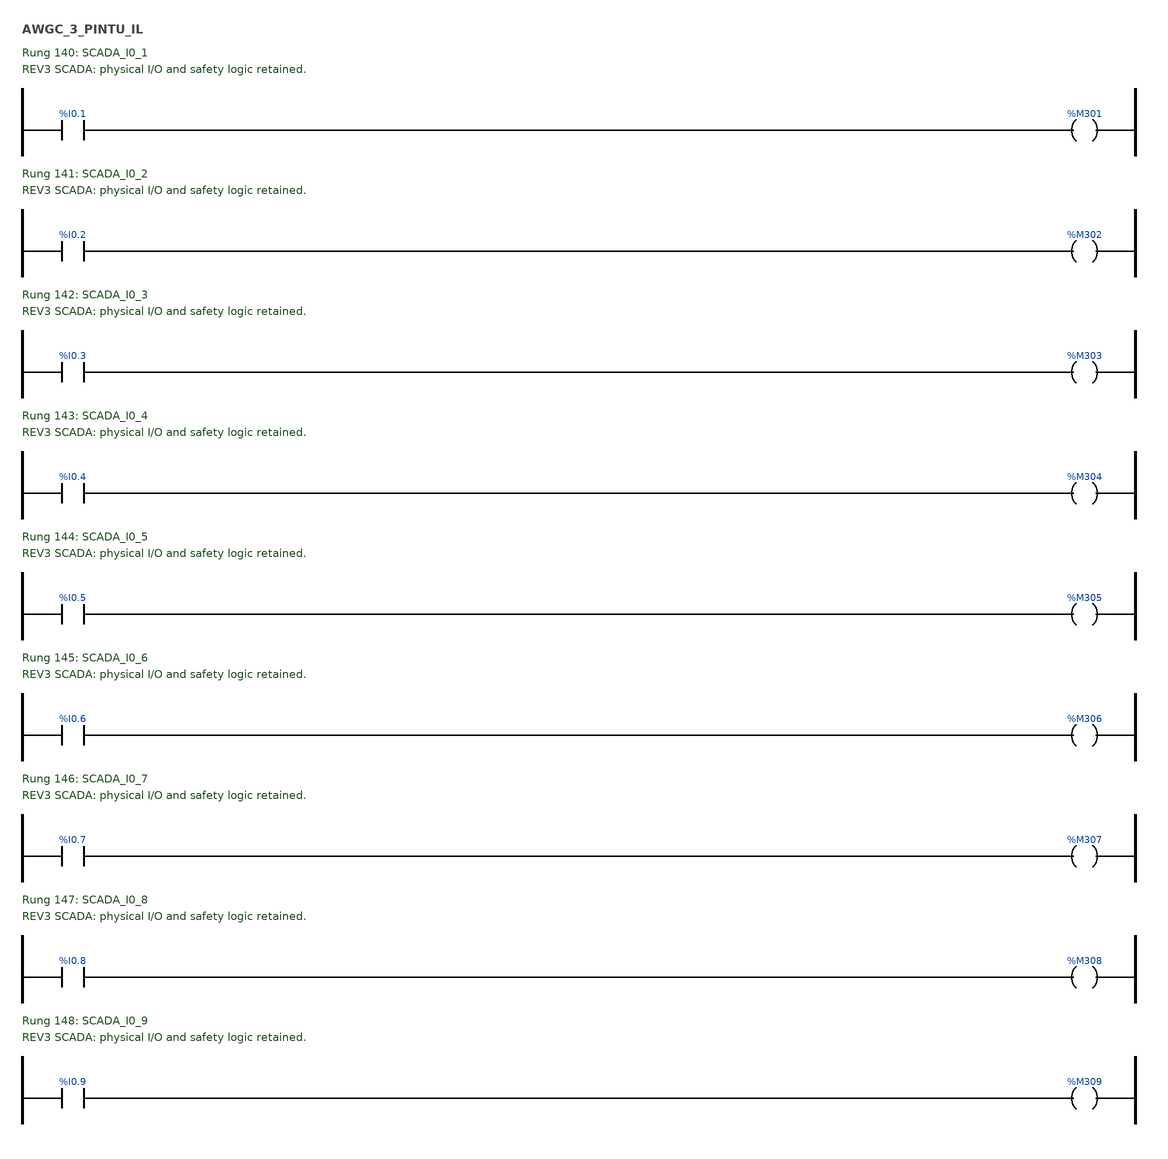

// Rung 140: SCADA_I0_1
// REV3 SCADA: physical I/O and safety logic retained.
  LD %I0.1                (* LS_CLOSE_G1 *)
  ST %M301                (* STATUS_I0_1 *)
  // as ST:
  //   STATUS_I0_1 := LS_CLOSE_G1;

// Rung 141: SCADA_I0_2
// REV3 SCADA: physical I/O and safety logic retained.
  LD %I0.2                (* LS_OPEN_G1 *)
  ST %M302                (* STATUS_I0_2 *)
  // as ST:
  //   STATUS_I0_2 := LS_OPEN_G1;

// Rung 142: SCADA_I0_3
// REV3 SCADA: physical I/O and safety logic retained.
  LD %I0.3                (* LS_CLOSE_G2 *)
  ST %M303                (* STATUS_I0_3 *)
  // as ST:
  //   STATUS_I0_3 := LS_CLOSE_G2;

// Rung 143: SCADA_I0_4
// REV3 SCADA: physical I/O and safety logic retained.
  LD %I0.4                (* LS_OPEN_G2 *)
  ST %M304                (* STATUS_I0_4 *)
  // as ST:
  //   STATUS_I0_4 := LS_OPEN_G2;

// Rung 144: SCADA_I0_5
// REV3 SCADA: physical I/O and safety logic retained.
  LD %I0.5                (* LS_CLOSE_G3 *)
  ST %M305                (* STATUS_I0_5 *)
  // as ST:
  //   STATUS_I0_5 := LS_CLOSE_G3;

// Rung 145: SCADA_I0_6
// REV3 SCADA: physical I/O and safety logic retained.
  LD %I0.6                (* LS_OPEN_G3 *)
  ST %M306                (* STATUS_I0_6 *)
  // as ST:
  //   STATUS_I0_6 := LS_OPEN_G3;

// Rung 146: SCADA_I0_7
// REV3 SCADA: physical I/O and safety logic retained.
  LD %I0.7                (* OL_OK_G1 *)
  ST %M307                (* STATUS_I0_7 *)
  // as ST:
  //   STATUS_I0_7 := OL_OK_G1;

// Rung 147: SCADA_I0_8
// REV3 SCADA: physical I/O and safety logic retained.
  LD %I0.8                (* OL_OK_G2 *)
  ST %M308                (* STATUS_I0_8 *)
  // as ST:
  //   STATUS_I0_8 := OL_OK_G2;

// Rung 148: SCADA_I0_9
// REV3 SCADA: physical I/O and safety logic retained.
  LD %I0.9                (* OL_OK_G3 *)
  ST %M309                (* STATUS_I0_9 *)
  // as ST:
  //   STATUS_I0_9 := OL_OK_G3;

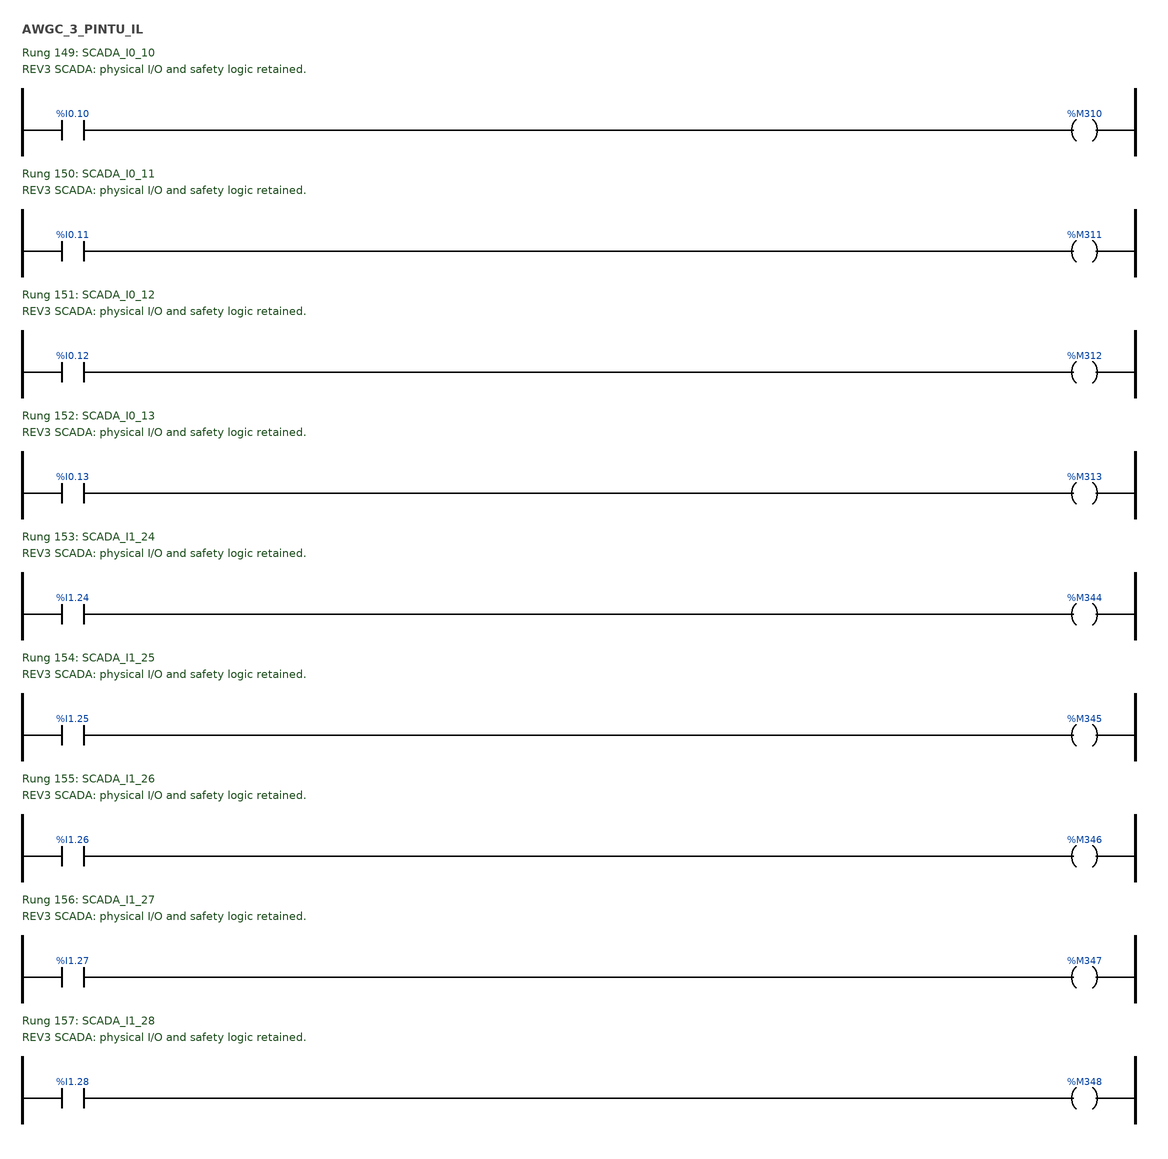

// Rung 149: SCADA_I0_10
// REV3 SCADA: physical I/O and safety logic retained.
  LD %I0.10               (* SPARE_I010 *)
  ST %M310                (* STATUS_I0_10 *)
  // as ST:
  //   STATUS_I0_10 := SPARE_I010;

// Rung 150: SCADA_I0_11
// REV3 SCADA: physical I/O and safety logic retained.
  LD %I0.11               (* SPARE_I011 *)
  ST %M311                (* STATUS_I0_11 *)
  // as ST:
  //   STATUS_I0_11 := SPARE_I011;

// Rung 151: SCADA_I0_12
// REV3 SCADA: physical I/O and safety logic retained.
  LD %I0.12               (* SPARE_I012 *)
  ST %M312                (* STATUS_I0_12 *)
  // as ST:
  //   STATUS_I0_12 := SPARE_I012;

// Rung 152: SCADA_I0_13
// REV3 SCADA: physical I/O and safety logic retained.
  LD %I0.13               (* SPARE_I013 *)
  ST %M313                (* STATUS_I0_13 *)
  // as ST:
  //   STATUS_I0_13 := SPARE_I013;

// Rung 153: SCADA_I1_24
// REV3 SCADA: physical I/O and safety logic retained.
  LD %I1.24               (* MODE_AUTO *)
  ST %M344                (* STATUS_I1_24 *)
  // as ST:
  //   STATUS_I1_24 := MODE_AUTO;

// Rung 154: SCADA_I1_25
// REV3 SCADA: physical I/O and safety logic retained.
  LD %I1.25               (* MAN_OPEN_G1 *)
  ST %M345                (* STATUS_I1_25 *)
  // as ST:
  //   STATUS_I1_25 := MAN_OPEN_G1;

// Rung 155: SCADA_I1_26
// REV3 SCADA: physical I/O and safety logic retained.
  LD %I1.26               (* MAN_CLOSE_G1 *)
  ST %M346                (* STATUS_I1_26 *)
  // as ST:
  //   STATUS_I1_26 := MAN_CLOSE_G1;

// Rung 156: SCADA_I1_27
// REV3 SCADA: physical I/O and safety logic retained.
  LD %I1.27               (* MAN_OPEN_G2 *)
  ST %M347                (* STATUS_I1_27 *)
  // as ST:
  //   STATUS_I1_27 := MAN_OPEN_G2;

// Rung 157: SCADA_I1_28
// REV3 SCADA: physical I/O and safety logic retained.
  LD %I1.28               (* MAN_CLOSE_G2 *)
  ST %M348                (* STATUS_I1_28 *)
  // as ST:
  //   STATUS_I1_28 := MAN_CLOSE_G2;

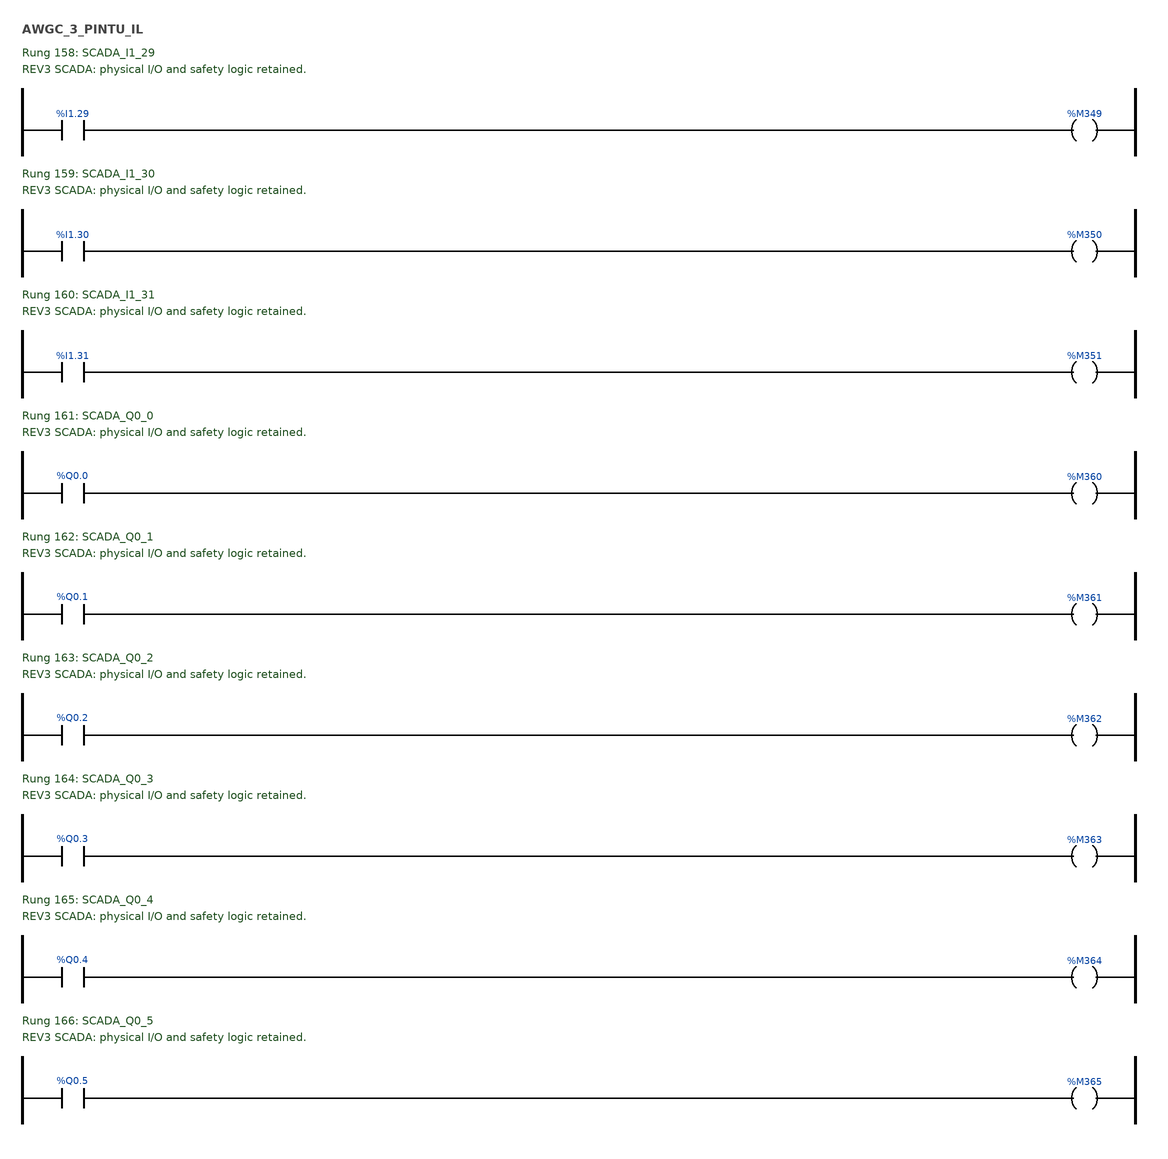

// Rung 158: SCADA_I1_29
// REV3 SCADA: physical I/O and safety logic retained.
  LD %I1.29               (* MAN_OPEN_G3 *)
  ST %M349                (* STATUS_I1_29 *)
  // as ST:
  //   STATUS_I1_29 := MAN_OPEN_G3;

// Rung 159: SCADA_I1_30
// REV3 SCADA: physical I/O and safety logic retained.
  LD %I1.30               (* MAN_CLOSE_G3 *)
  ST %M350                (* STATUS_I1_30 *)
  // as ST:
  //   STATUS_I1_30 := MAN_CLOSE_G3;

// Rung 160: SCADA_I1_31
// REV3 SCADA: physical I/O and safety logic retained.
  LD %I1.31               (* RESET_FAULT *)
  ST %M351                (* STATUS_I1_31 *)
  // as ST:
  //   STATUS_I1_31 := RESET_FAULT;

// Rung 161: SCADA_Q0_0
// REV3 SCADA: physical I/O and safety logic retained.
  LD %Q0.0                (* OPEN_G1 *)
  ST %M360                (* STATUS_Q0_0 *)
  // as ST:
  //   STATUS_Q0_0 := OPEN_G1;

// Rung 162: SCADA_Q0_1
// REV3 SCADA: physical I/O and safety logic retained.
  LD %Q0.1                (* CLOSE_G1 *)
  ST %M361                (* STATUS_Q0_1 *)
  // as ST:
  //   STATUS_Q0_1 := CLOSE_G1;

// Rung 163: SCADA_Q0_2
// REV3 SCADA: physical I/O and safety logic retained.
  LD %Q0.2                (* OPEN_G2 *)
  ST %M362                (* STATUS_Q0_2 *)
  // as ST:
  //   STATUS_Q0_2 := OPEN_G2;

// Rung 164: SCADA_Q0_3
// REV3 SCADA: physical I/O and safety logic retained.
  LD %Q0.3                (* CLOSE_G2 *)
  ST %M363                (* STATUS_Q0_3 *)
  // as ST:
  //   STATUS_Q0_3 := CLOSE_G2;

// Rung 165: SCADA_Q0_4
// REV3 SCADA: physical I/O and safety logic retained.
  LD %Q0.4                (* OPEN_G3 *)
  ST %M364                (* STATUS_Q0_4 *)
  // as ST:
  //   STATUS_Q0_4 := OPEN_G3;

// Rung 166: SCADA_Q0_5
// REV3 SCADA: physical I/O and safety logic retained.
  LD %Q0.5                (* CLOSE_G3 *)
  ST %M365                (* STATUS_Q0_5 *)
  // as ST:
  //   STATUS_Q0_5 := CLOSE_G3;
